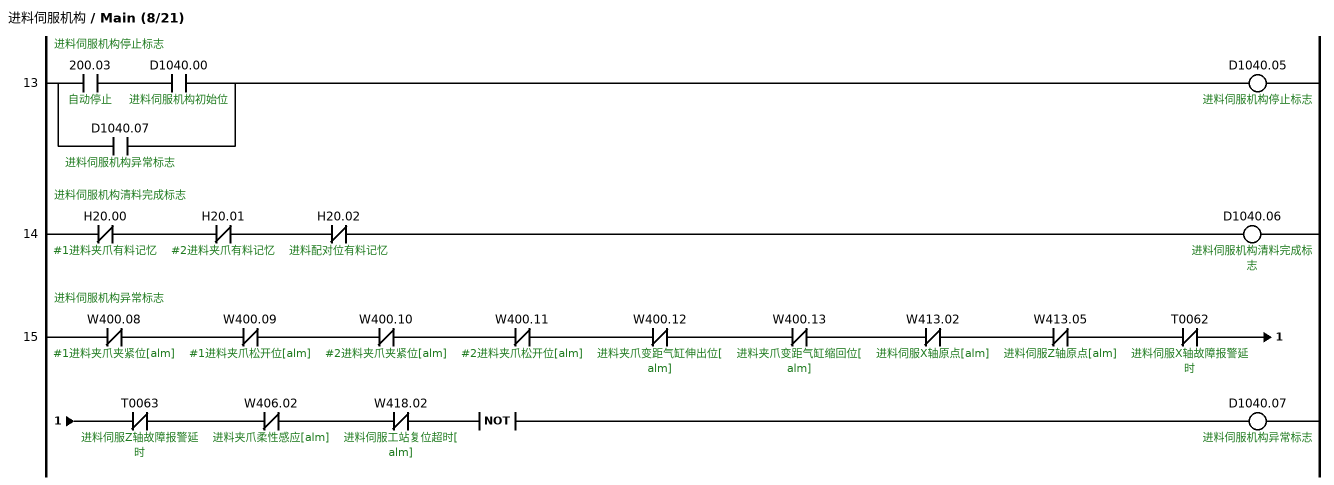
; [picture p72: 进料伺服机构 / Main, rungs 13-15]
; rung 13: 进料伺服机构停止标志
LD 200.03  ; 自动停止
AND D1040.00  ; 进料伺服机构初始位
OR D1040.07  ; 进料伺服机构异常标志
OUT D1040.05  ; 进料伺服机构停止标志
; rung 14: 进料伺服机构清料完成标志
LDNOT H20.00  ; #1进料夹爪有料记忆
ANDNOT H20.01  ; #2进料夹爪有料记忆
ANDNOT H20.02  ; 进料配对位有料记忆
OUT D1040.06  ; 进料伺服机构清料完成标志
; rung 15: 进料伺服机构异常标志
LDNOT W400.08  ; #1进料夹爪夹紧位[alm]
ANDNOT W400.09  ; #1进料夹爪松开位[alm]
ANDNOT W400.10  ; #2进料夹爪夹紧位[alm]
ANDNOT W400.11  ; #2进料夹爪松开位[alm]
ANDNOT W400.12  ; 进料夹爪变距气缸伸出位[alm]
ANDNOT W400.13  ; 进料夹爪变距气缸缩回位[alm]
ANDNOT W413.02  ; 进料伺服X轴原点[alm]
ANDNOT W413.05  ; 进料伺服Z轴原点[alm]
ANDNOT T0062  ; 进料伺服X轴故障报警延时
ANDNOT T0063  ; 进料伺服Z轴故障报警延时
ANDNOT W406.02  ; 进料夹爪柔性感应[alm]
ANDNOT W418.02  ; 进料伺服工站复位超时[alm]
NOT(520)
OUT D1040.07  ; 进料伺服机构异常标志

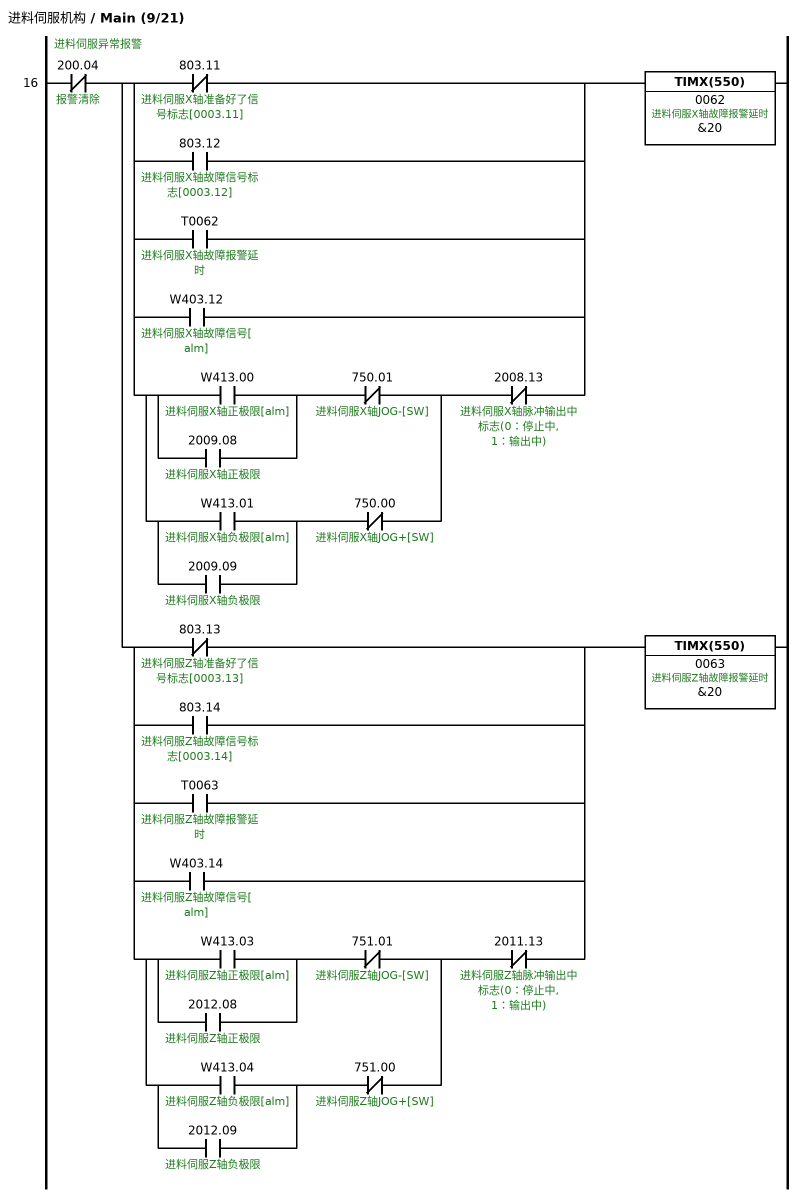
; rung 16: 进料伺服异常报警
LDNOT 200.04  ; 报警清除
OUT TR0
LDNOT 803.11  ; 进料伺服X轴准备好了信号标志[0003.11]
OR 803.12  ; 进料伺服X轴故障信号标志[0003.12]
OR T0062  ; 进料伺服X轴故障报警延时
OR W403.12  ; 进料伺服X轴故障信号[alm]
LD W413.00  ; 进料伺服X轴正极限[alm]
OR 2009.08  ; 进料伺服X轴正极限
ANDNOT 750.01  ; 进料伺服X轴JOG-[SW]
LD W413.01  ; 进料伺服X轴负极限[alm]
OR 2009.09  ; 进料伺服X轴负极限
ANDNOT 750.00  ; 进料伺服X轴JOG+[SW]
ORLD
ANDNOT 2008.13  ; 进料伺服X轴脉冲输出中标志(0：停止中,1：输出中)
ORLD
ANDLD
TIMX(550) 0062 &20  ; 进料伺服X轴故障报警延时
LD TR0
LDNOT 803.13  ; 进料伺服Z轴准备好了信号标志[0003.13]
OR 803.14  ; 进料伺服Z轴故障信号标志[0003.14]
OR T0063  ; 进料伺服Z轴故障报警延时
OR W403.14  ; 进料伺服Z轴故障信号[alm]
LD W413.03  ; 进料伺服Z轴正极限[alm]
OR 2012.08  ; 进料伺服Z轴正极限
ANDNOT 751.01  ; 进料伺服Z轴JOG-[SW]
LD W413.04  ; 进料伺服Z轴负极限[alm]
OR 2012.09  ; 进料伺服Z轴负极限
ANDNOT 751.00  ; 进料伺服Z轴JOG+[SW]
ORLD
ANDNOT 2011.13  ; 进料伺服Z轴脉冲输出中标志(0：停止中,1：输出中)
ORLD
ANDLD
TIMX(550) 0063 &20  ; 进料伺服Z轴故障报警延时

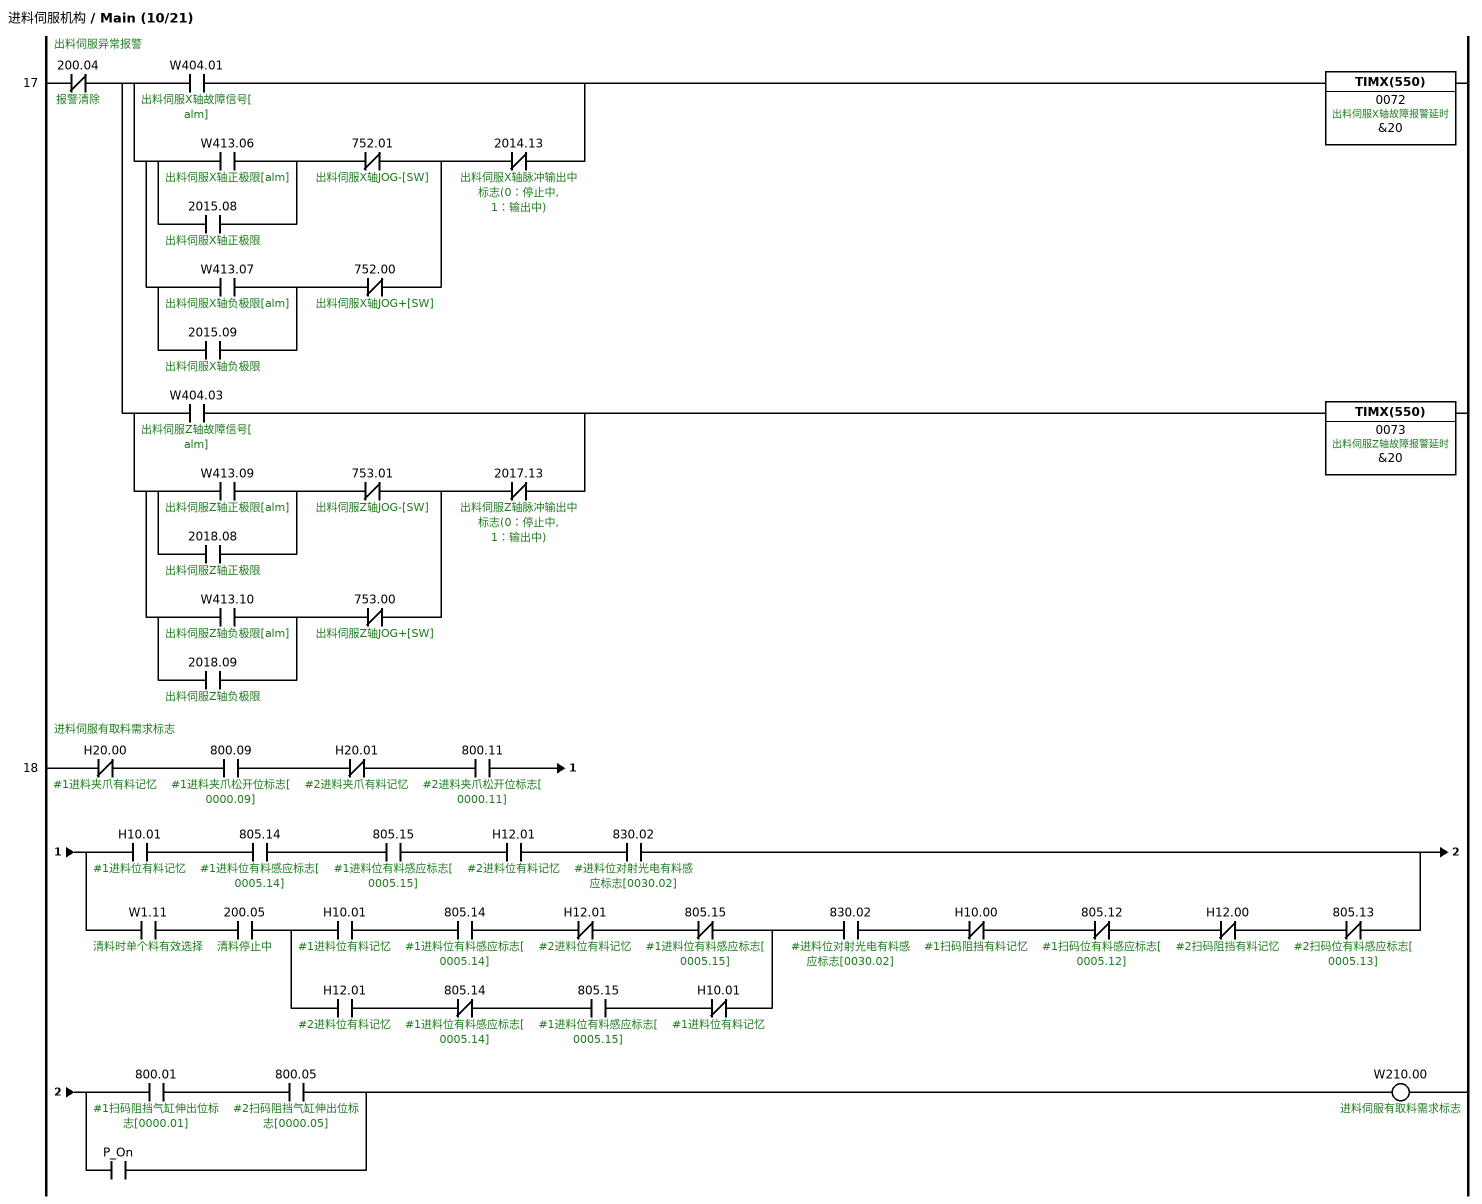
; rung 17: 出料伺服异常报警
LDNOT 200.04  ; 报警清除
OUT TR0
LD W404.01  ; 出料伺服X轴故障信号[alm]
LD W413.06  ; 出料伺服X轴正极限[alm]
OR 2015.08  ; 出料伺服X轴正极限
ANDNOT 752.01  ; 出料伺服X轴JOG-[SW]
LD W413.07  ; 出料伺服X轴负极限[alm]
OR 2015.09  ; 出料伺服X轴负极限
ANDNOT 752.00  ; 出料伺服X轴JOG+[SW]
ORLD
ANDNOT 2014.13  ; 出料伺服X轴脉冲输出中标志(0：停止中,1：输出中)
ORLD
ANDLD
TIMX(550) 0072 &20  ; 出料伺服X轴故障报警延时
LD TR0
LD W404.03  ; 出料伺服Z轴故障信号[alm]
LD W413.09  ; 出料伺服Z轴正极限[alm]
OR 2018.08  ; 出料伺服Z轴正极限
ANDNOT 753.01  ; 出料伺服Z轴JOG-[SW]
LD W413.10  ; 出料伺服Z轴负极限[alm]
OR 2018.09  ; 出料伺服Z轴负极限
ANDNOT 753.00  ; 出料伺服Z轴JOG+[SW]
ORLD
ANDNOT 2017.13  ; 出料伺服Z轴脉冲输出中标志(0：停止中,1：输出中)
ORLD
ANDLD
TIMX(550) 0073 &20  ; 出料伺服Z轴故障报警延时
; rung 18: 进料伺服有取料需求标志
LDNOT H20.00  ; #1进料夹爪有料记忆
AND 800.09  ; #1进料夹爪松开位标志[0000.09]
ANDNOT H20.01  ; #2进料夹爪有料记忆
AND 800.11  ; #2进料夹爪松开位标志[0000.11]
LD H10.01  ; #1进料位有料记忆
AND 805.14  ; #1进料位有料感应标志[0005.14]
AND 805.15  ; #1进料位有料感应标志[0005.15]
AND H12.01  ; #2进料位有料记忆
AND 830.02  ; #进料位对射光电有料感应标志[0030.02]
LD W1.11  ; 清料时单个料有效选择
AND 200.05  ; 清料停止中
LD H10.01  ; #1进料位有料记忆
AND 805.14  ; #1进料位有料感应标志[0005.14]
ANDNOT H12.01  ; #2进料位有料记忆
ANDNOT 805.15  ; #1进料位有料感应标志[0005.15]
LD H12.01  ; #2进料位有料记忆
ANDNOT 805.14  ; #1进料位有料感应标志[0005.14]
AND 805.15  ; #1进料位有料感应标志[0005.15]
ANDNOT H10.01  ; #1进料位有料记忆
ORLD
ANDLD
AND 830.02  ; #进料位对射光电有料感应标志[0030.02]
ANDNOT H10.00  ; #1扫码阻挡有料记忆
ANDNOT 805.12  ; #1扫码位有料感应标志[0005.12]
ANDNOT H12.00  ; #2扫码阻挡有料记忆
ANDNOT 805.13  ; #2扫码位有料感应标志[0005.13]
ORLD
ANDLD
LD 800.01  ; #1扫码阻挡气缸伸出位标志[0000.01]
AND 800.05  ; #2扫码阻挡气缸伸出位标志[0000.05]
OR P_On
ANDLD
OUT W210.00  ; 进料伺服有取料需求标志

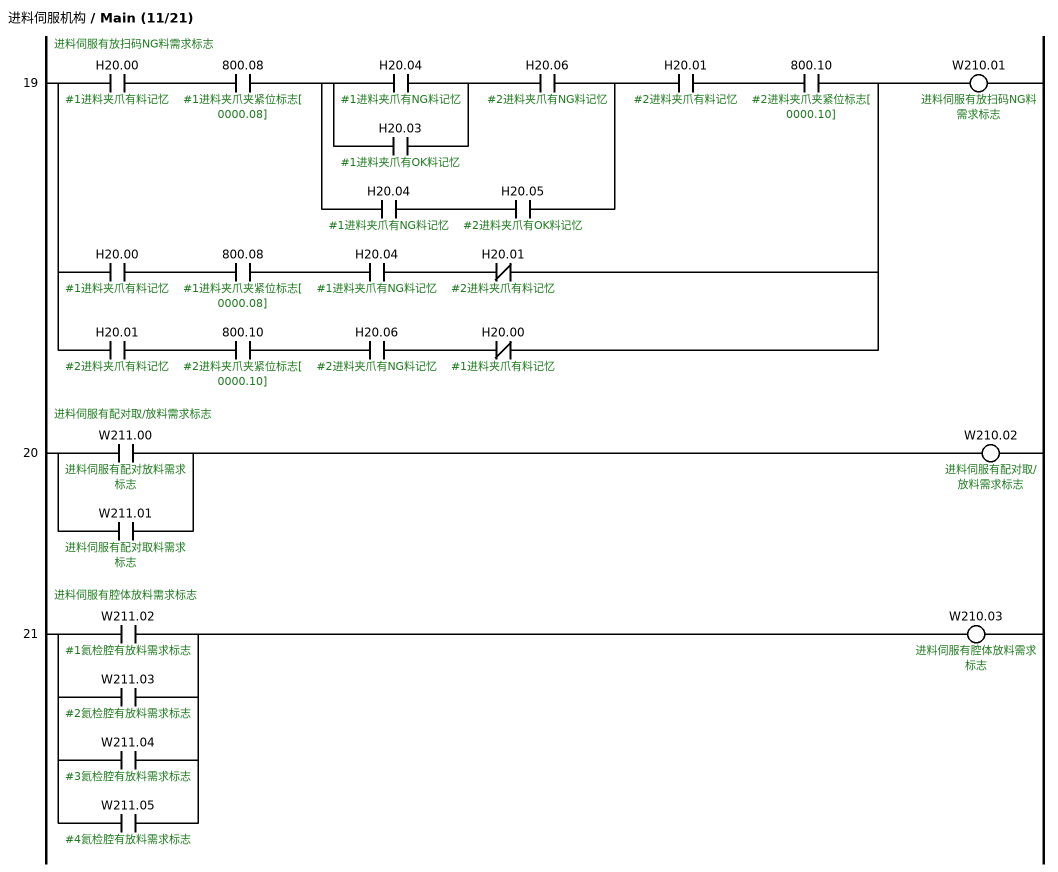
; rung 19: 进料伺服有放扫码NG料需求标志
LD H20.00  ; #1进料夹爪有料记忆
AND 800.08  ; #1进料夹爪夹紧位标志[0000.08]
LD H20.04  ; #1进料夹爪有NG料记忆
OR H20.03  ; #1进料夹爪有OK料记忆
AND H20.06  ; #2进料夹爪有NG料记忆
LD H20.04  ; #1进料夹爪有NG料记忆
AND H20.05  ; #2进料夹爪有OK料记忆
ORLD
ANDLD
AND H20.01  ; #2进料夹爪有料记忆
AND 800.10  ; #2进料夹爪夹紧位标志[0000.10]
LD H20.00  ; #1进料夹爪有料记忆
AND 800.08  ; #1进料夹爪夹紧位标志[0000.08]
AND H20.04  ; #1进料夹爪有NG料记忆
ANDNOT H20.01  ; #2进料夹爪有料记忆
ORLD
LD H20.01  ; #2进料夹爪有料记忆
AND 800.10  ; #2进料夹爪夹紧位标志[0000.10]
AND H20.06  ; #2进料夹爪有NG料记忆
ANDNOT H20.00  ; #1进料夹爪有料记忆
ORLD
OUT W210.01  ; 进料伺服有放扫码NG料需求标志
; rung 20: 进料伺服有配对取/放料需求标志
LD W211.00  ; 进料伺服有配对放料需求标志
OR W211.01  ; 进料伺服有配对取料需求标志
OUT W210.02  ; 进料伺服有配对取/放料需求标志
; rung 21: 进料伺服有腔体放料需求标志
LD W211.02  ; #1氦检腔有放料需求标志
OR W211.03  ; #2氦检腔有放料需求标志
OR W211.04  ; #3氦检腔有放料需求标志
OR W211.05  ; #4氦检腔有放料需求标志
OUT W210.03  ; 进料伺服有腔体放料需求标志

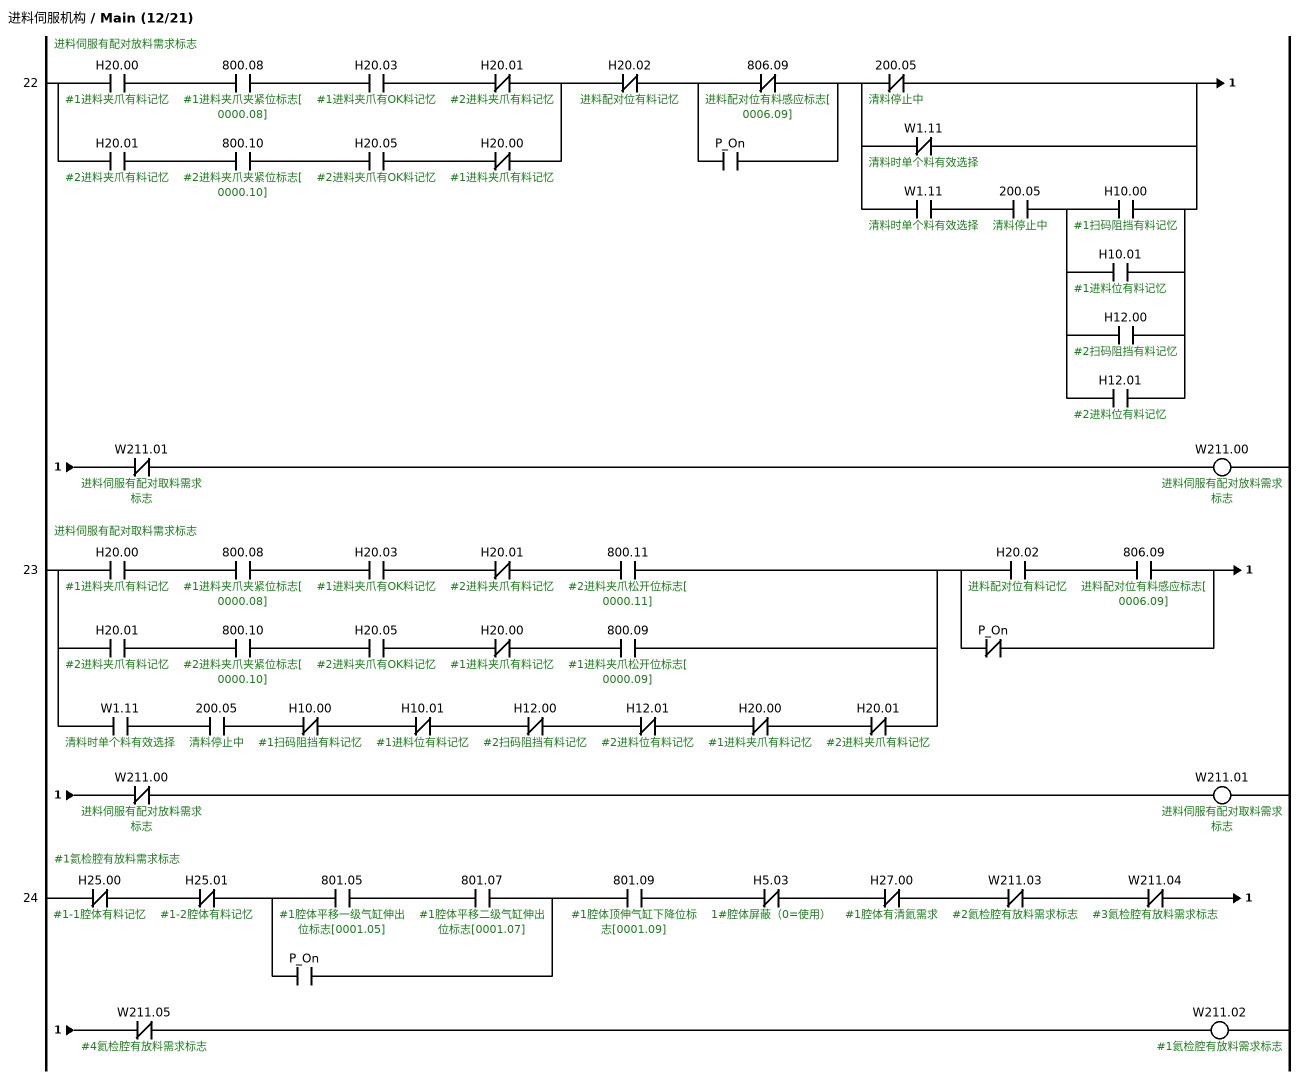
; rung 22: 进料伺服有配对放料需求标志
LD H20.00  ; #1进料夹爪有料记忆
AND 800.08  ; #1进料夹爪夹紧位标志[0000.08]
AND H20.03  ; #1进料夹爪有OK料记忆
ANDNOT H20.01  ; #2进料夹爪有料记忆
LD H20.01  ; #2进料夹爪有料记忆
AND 800.10  ; #2进料夹爪夹紧位标志[0000.10]
AND H20.05  ; #2进料夹爪有OK料记忆
ANDNOT H20.00  ; #1进料夹爪有料记忆
ORLD
ANDNOT H20.02  ; 进料配对位有料记忆
LDNOT 806.09  ; 进料配对位有料感应标志[0006.09]
OR P_On
ANDLD
LDNOT 200.05  ; 清料停止中
ORNOT W1.11  ; 清料时单个料有效选择
LD W1.11  ; 清料时单个料有效选择
AND 200.05  ; 清料停止中
LD H10.00  ; #1扫码阻挡有料记忆
OR H10.01  ; #1进料位有料记忆
OR H12.00  ; #2扫码阻挡有料记忆
OR H12.01  ; #2进料位有料记忆
ANDLD
ORLD
ANDLD
ANDNOT W211.01  ; 进料伺服有配对取料需求标志
OUT W211.00  ; 进料伺服有配对放料需求标志
; rung 23: 进料伺服有配对取料需求标志
LD H20.00  ; #1进料夹爪有料记忆
AND 800.08  ; #1进料夹爪夹紧位标志[0000.08]
AND H20.03  ; #1进料夹爪有OK料记忆
ANDNOT H20.01  ; #2进料夹爪有料记忆
AND 800.11  ; #2进料夹爪松开位标志[0000.11]
LD H20.01  ; #2进料夹爪有料记忆
AND 800.10  ; #2进料夹爪夹紧位标志[0000.10]
AND H20.05  ; #2进料夹爪有OK料记忆
ANDNOT H20.00  ; #1进料夹爪有料记忆
AND 800.09  ; #1进料夹爪松开位标志[0000.09]
ORLD
LD W1.11  ; 清料时单个料有效选择
AND 200.05  ; 清料停止中
ANDNOT H10.00  ; #1扫码阻挡有料记忆
ANDNOT H10.01  ; #1进料位有料记忆
ANDNOT H12.00  ; #2扫码阻挡有料记忆
ANDNOT H12.01  ; #2进料位有料记忆
ANDNOT H20.00  ; #1进料夹爪有料记忆
ANDNOT H20.01  ; #2进料夹爪有料记忆
ORLD
LD H20.02  ; 进料配对位有料记忆
AND 806.09  ; 进料配对位有料感应标志[0006.09]
ORNOT P_On
ANDLD
ANDNOT W211.00  ; 进料伺服有配对放料需求标志
OUT W211.01  ; 进料伺服有配对取料需求标志
; rung 24: #1氦检腔有放料需求标志
LDNOT H25.00  ; #1-1腔体有料记忆
ANDNOT H25.01  ; #1-2腔体有料记忆
LD 801.05  ; #1腔体平移一级气缸伸出位标志[0001.05]
AND 801.07  ; #1腔体平移二级气缸伸出位标志[0001.07]
OR P_On
ANDLD
AND 801.09  ; #1腔体顶伸气缸下降位标志[0001.09]
ANDNOT H5.03  ; 1#腔体屏蔽（0=使用）
ANDNOT H27.00  ; #1腔体有清氦需求
ANDNOT W211.03  ; #2氦检腔有放料需求标志
ANDNOT W211.04  ; #3氦检腔有放料需求标志
ANDNOT W211.05  ; #4氦检腔有放料需求标志
OUT W211.02  ; #1氦检腔有放料需求标志

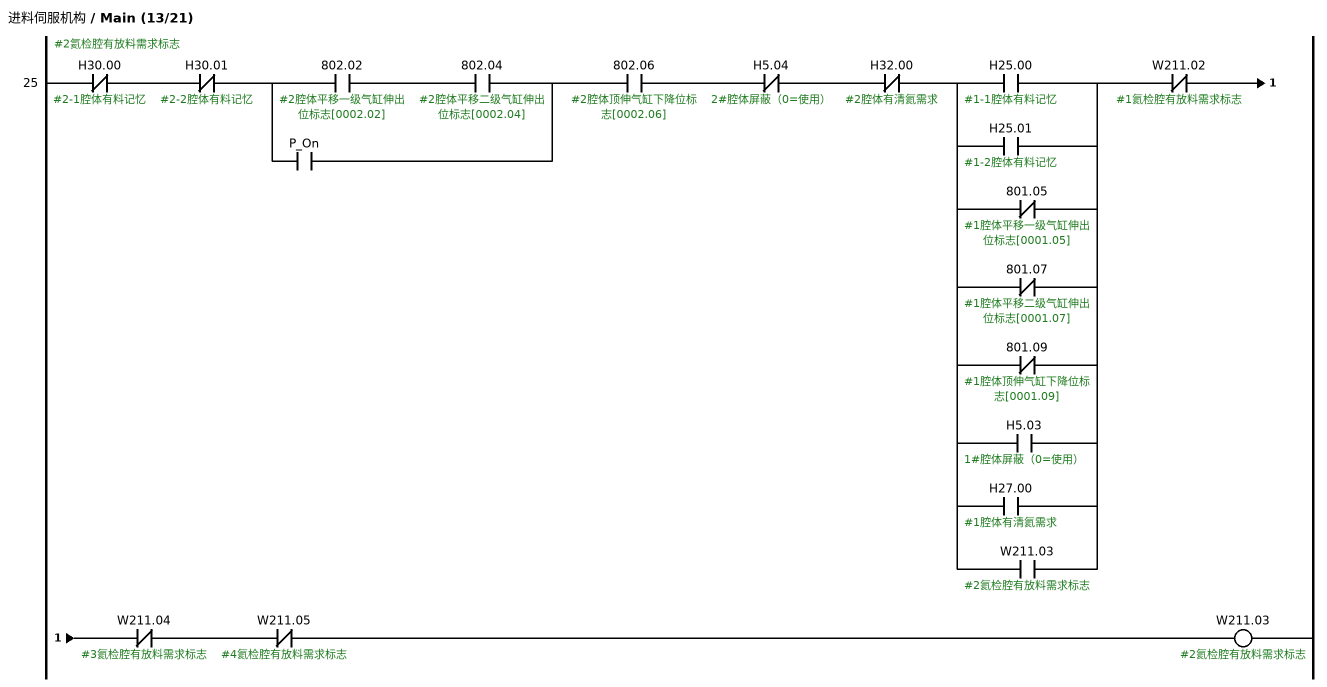
; rung 25: #2氦检腔有放料需求标志
LDNOT H30.00  ; #2-1腔体有料记忆
ANDNOT H30.01  ; #2-2腔体有料记忆
LD 802.02  ; #2腔体平移一级气缸伸出位标志[0002.02]
AND 802.04  ; #2腔体平移二级气缸伸出位标志[0002.04]
OR P_On
ANDLD
AND 802.06  ; #2腔体顶伸气缸下降位标志[0002.06]
ANDNOT H5.04  ; 2#腔体屏蔽（0=使用）
ANDNOT H32.00  ; #2腔体有清氦需求
LD H25.00  ; #1-1腔体有料记忆
OR H25.01  ; #1-2腔体有料记忆
ORNOT 801.05  ; #1腔体平移一级气缸伸出位标志[0001.05]
ORNOT 801.07  ; #1腔体平移二级气缸伸出位标志[0001.07]
ORNOT 801.09  ; #1腔体顶伸气缸下降位标志[0001.09]
OR H5.03  ; 1#腔体屏蔽（0=使用）
OR H27.00  ; #1腔体有清氦需求
OR W211.03  ; #2氦检腔有放料需求标志
ANDLD
ANDNOT W211.02  ; #1氦检腔有放料需求标志
ANDNOT W211.04  ; #3氦检腔有放料需求标志
ANDNOT W211.05  ; #4氦检腔有放料需求标志
OUT W211.03  ; #2氦检腔有放料需求标志

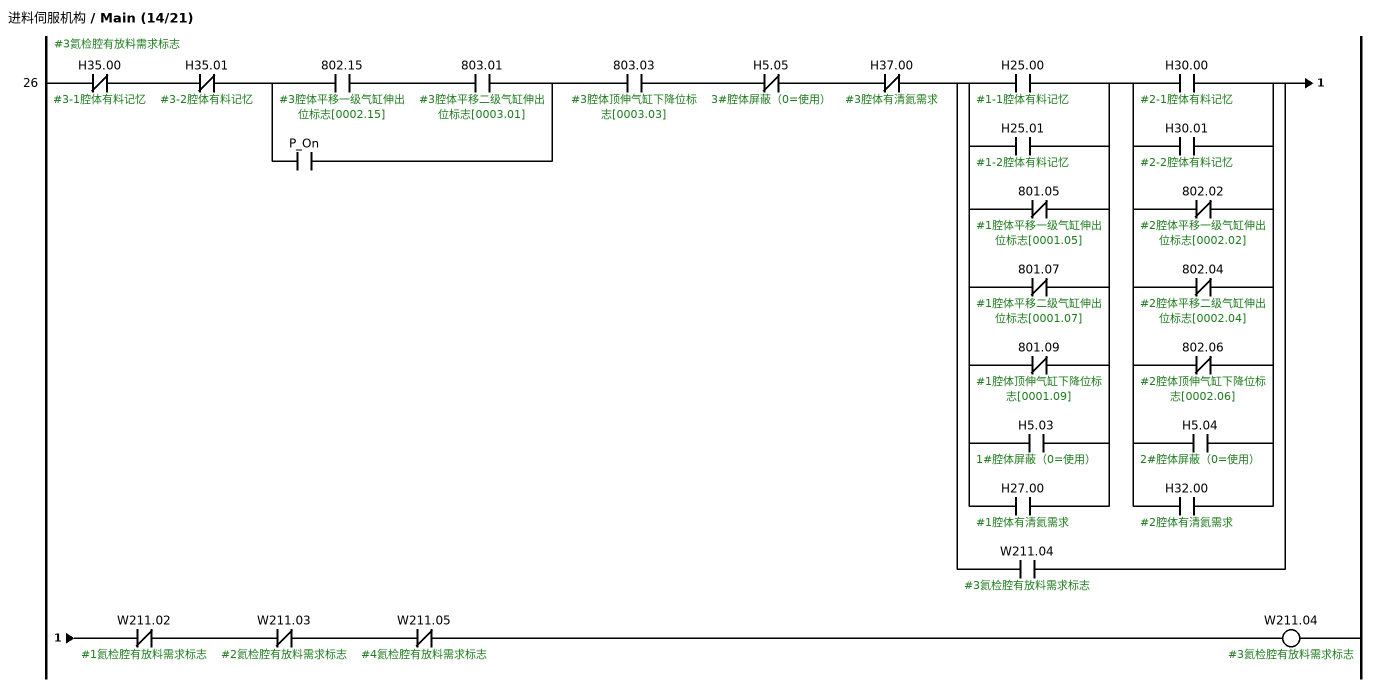
; rung 26: #3氦检腔有放料需求标志
LDNOT H35.00  ; #3-1腔体有料记忆
ANDNOT H35.01  ; #3-2腔体有料记忆
LD 802.15  ; #3腔体平移一级气缸伸出位标志[0002.15]
AND 803.01  ; #3腔体平移二级气缸伸出位标志[0003.01]
OR P_On
ANDLD
AND 803.03  ; #3腔体顶伸气缸下降位标志[0003.03]
ANDNOT H5.05  ; 3#腔体屏蔽（0=使用）
ANDNOT H37.00  ; #3腔体有清氦需求
LD H25.00  ; #1-1腔体有料记忆
OR H25.01  ; #1-2腔体有料记忆
ORNOT 801.05  ; #1腔体平移一级气缸伸出位标志[0001.05]
ORNOT 801.07  ; #1腔体平移二级气缸伸出位标志[0001.07]
ORNOT 801.09  ; #1腔体顶伸气缸下降位标志[0001.09]
OR H5.03  ; 1#腔体屏蔽（0=使用）
OR H27.00  ; #1腔体有清氦需求
LD H30.00  ; #2-1腔体有料记忆
OR H30.01  ; #2-2腔体有料记忆
ORNOT 802.02  ; #2腔体平移一级气缸伸出位标志[0002.02]
ORNOT 802.04  ; #2腔体平移二级气缸伸出位标志[0002.04]
ORNOT 802.06  ; #2腔体顶伸气缸下降位标志[0002.06]
OR H5.04  ; 2#腔体屏蔽（0=使用）
OR H32.00  ; #2腔体有清氦需求
ANDLD
OR W211.04  ; #3氦检腔有放料需求标志
ANDLD
ANDNOT W211.02  ; #1氦检腔有放料需求标志
ANDNOT W211.03  ; #2氦检腔有放料需求标志
ANDNOT W211.05  ; #4氦检腔有放料需求标志
OUT W211.04  ; #3氦检腔有放料需求标志

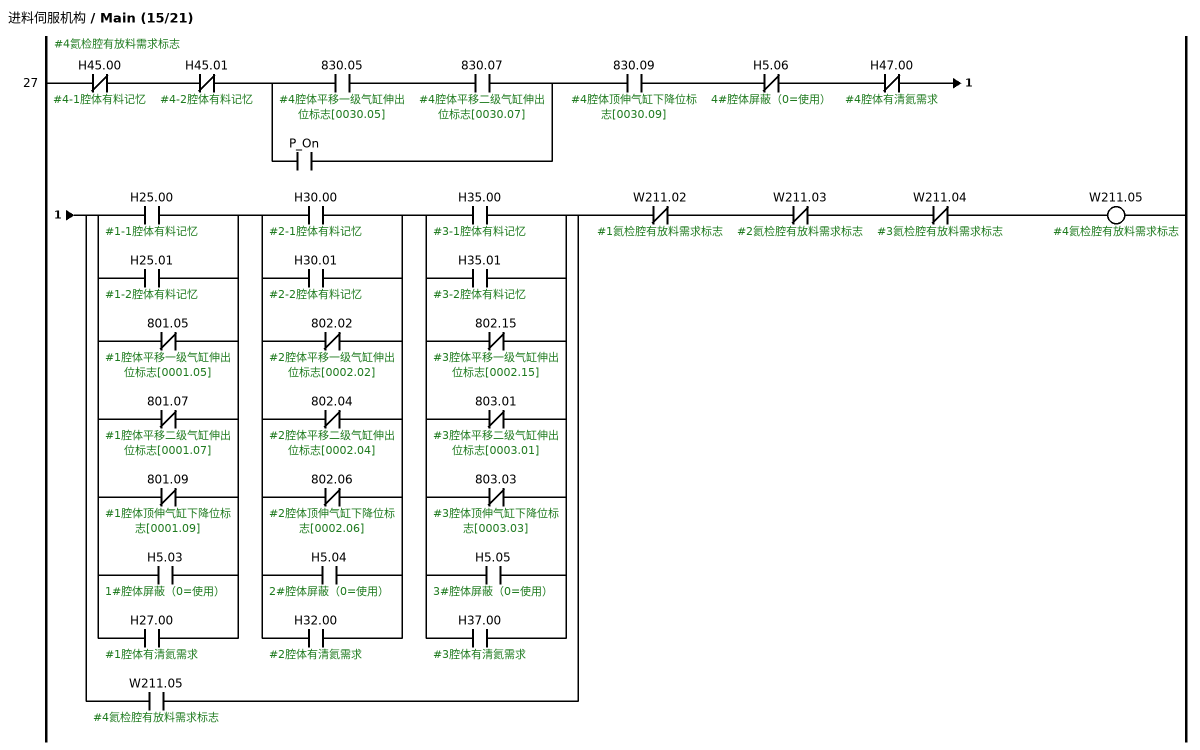
; rung 27: #4氦检腔有放料需求标志
LDNOT H45.00  ; #4-1腔体有料记忆
ANDNOT H45.01  ; #4-2腔体有料记忆
LD 830.05  ; #4腔体平移一级气缸伸出位标志[0030.05]
AND 830.07  ; #4腔体平移二级气缸伸出位标志[0030.07]
OR P_On
ANDLD
AND 830.09  ; #4腔体顶伸气缸下降位标志[0030.09]
ANDNOT H5.06  ; 4#腔体屏蔽（0=使用）
ANDNOT H47.00  ; #4腔体有清氦需求
LD H25.00  ; #1-1腔体有料记忆
OR H25.01  ; #1-2腔体有料记忆
ORNOT 801.05  ; #1腔体平移一级气缸伸出位标志[0001.05]
ORNOT 801.07  ; #1腔体平移二级气缸伸出位标志[0001.07]
ORNOT 801.09  ; #1腔体顶伸气缸下降位标志[0001.09]
OR H5.03  ; 1#腔体屏蔽（0=使用）
OR H27.00  ; #1腔体有清氦需求
LD H30.00  ; #2-1腔体有料记忆
OR H30.01  ; #2-2腔体有料记忆
ORNOT 802.02  ; #2腔体平移一级气缸伸出位标志[0002.02]
ORNOT 802.04  ; #2腔体平移二级气缸伸出位标志[0002.04]
ORNOT 802.06  ; #2腔体顶伸气缸下降位标志[0002.06]
OR H5.04  ; 2#腔体屏蔽（0=使用）
OR H32.00  ; #2腔体有清氦需求
ANDLD
LD H35.00  ; #3-1腔体有料记忆
OR H35.01  ; #3-2腔体有料记忆
ORNOT 802.15  ; #3腔体平移一级气缸伸出位标志[0002.15]
ORNOT 803.01  ; #3腔体平移二级气缸伸出位标志[0003.01]
ORNOT 803.03  ; #3腔体顶伸气缸下降位标志[0003.03]
OR H5.05  ; 3#腔体屏蔽（0=使用）
OR H37.00  ; #3腔体有清氦需求
ANDLD
OR W211.05  ; #4氦检腔有放料需求标志
ANDLD
ANDNOT W211.02  ; #1氦检腔有放料需求标志
ANDNOT W211.03  ; #2氦检腔有放料需求标志
ANDNOT W211.04  ; #3氦检腔有放料需求标志
OUT W211.05  ; #4氦检腔有放料需求标志

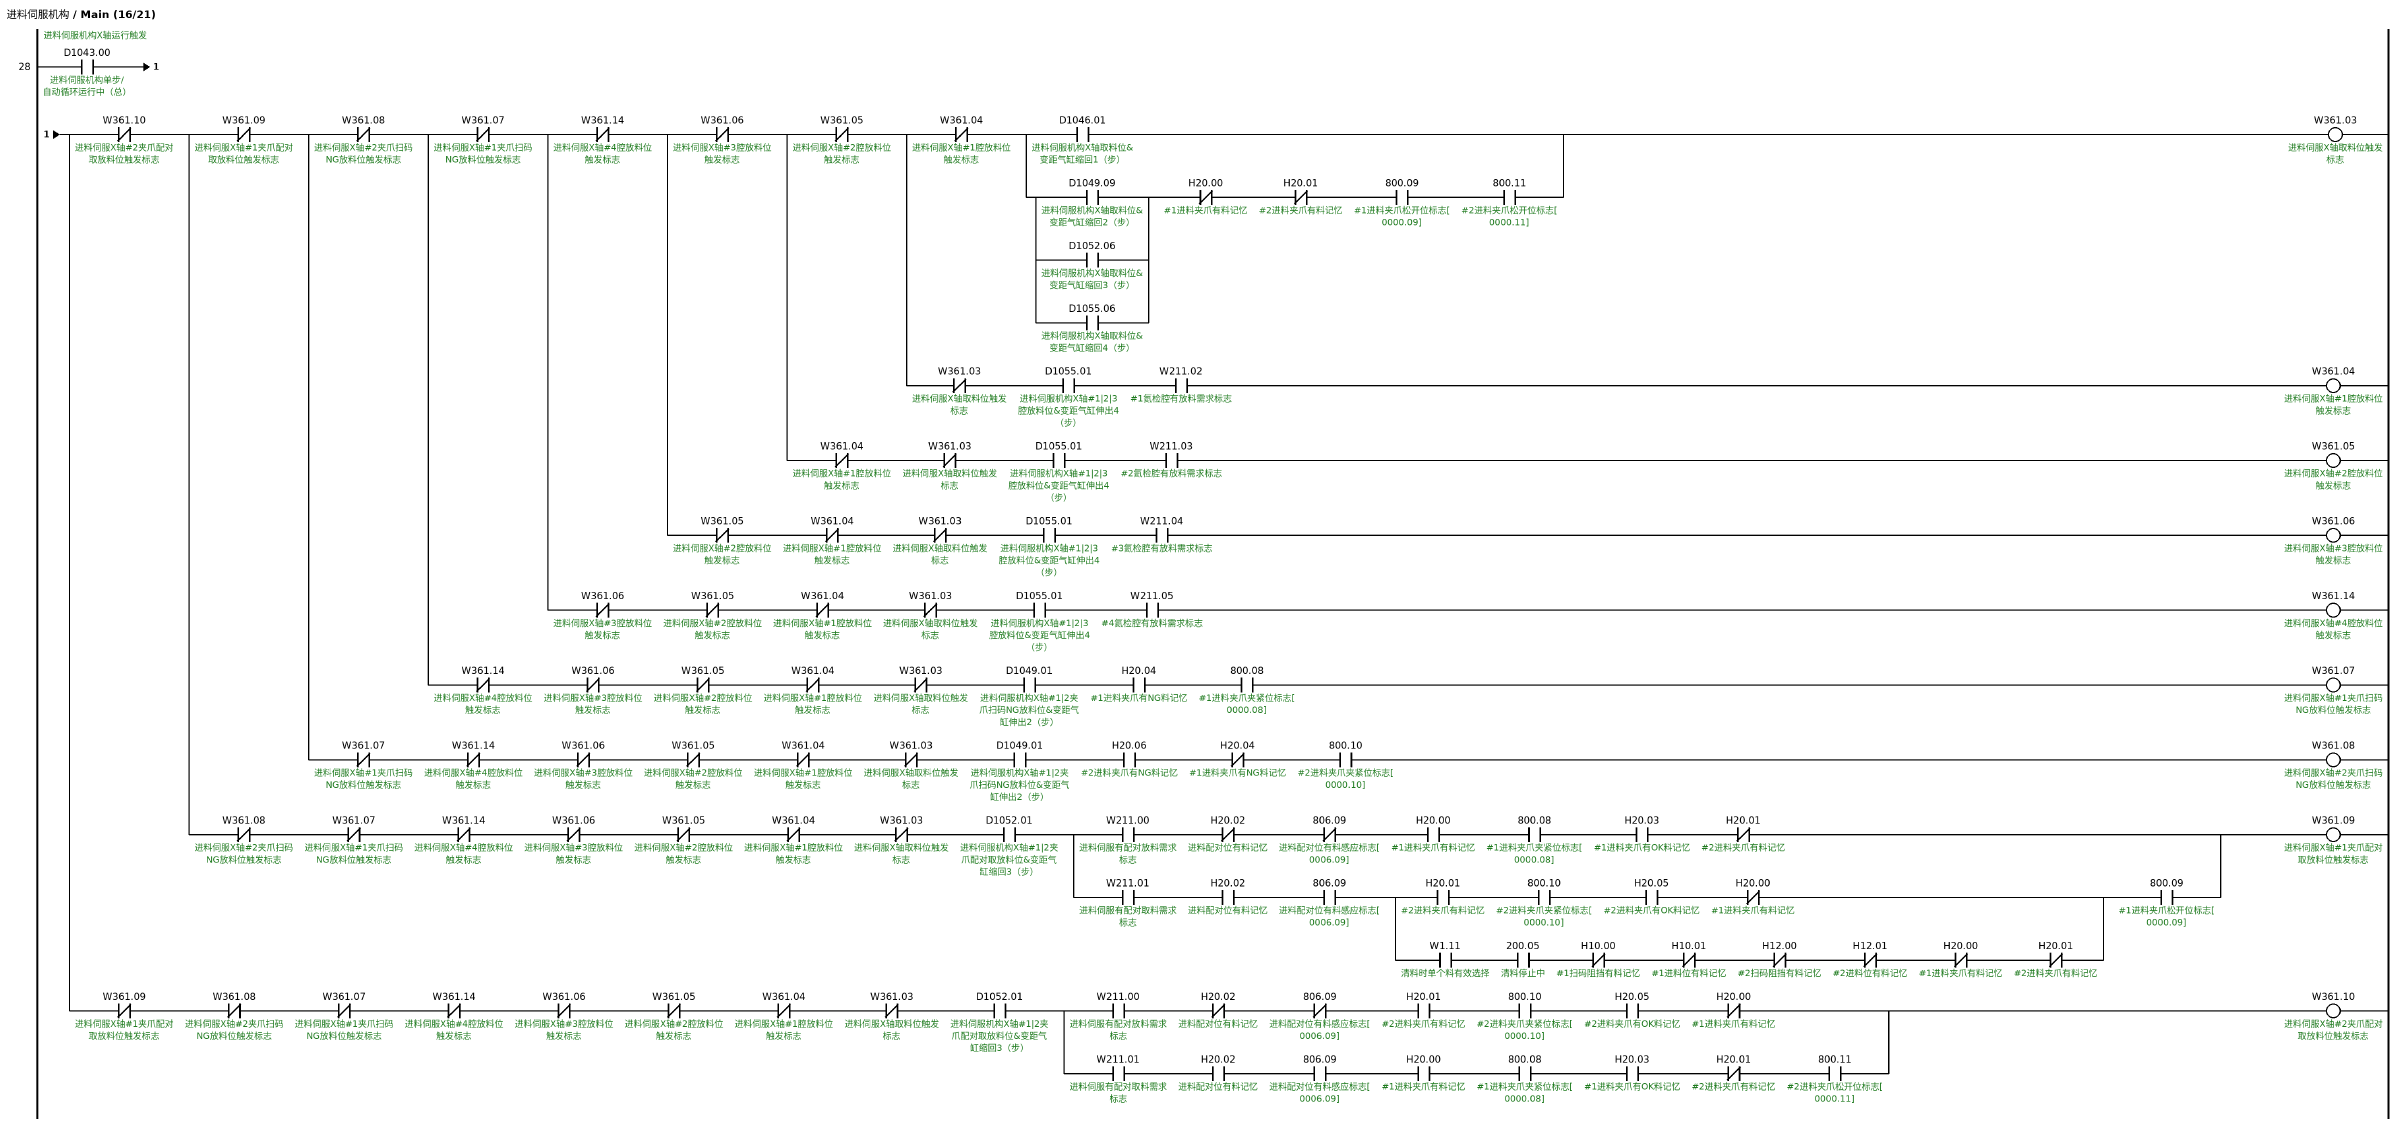
; rung 28: 进料伺服机构X轴运行触发
LD D1043.00  ; 进料伺服机构单步/自动循环运行中（总）
OUT TR0
ANDNOT W361.10  ; 进料伺服X轴#2夹爪配对取放料位触发标志
OUT TR1
ANDNOT W361.09  ; 进料伺服X轴#1夹爪配对取放料位触发标志
OUT TR2
ANDNOT W361.08  ; 进料伺服X轴#2夹爪扫码NG放料位触发标志
OUT TR3
ANDNOT W361.07  ; 进料伺服X轴#1夹爪扫码NG放料位触发标志
OUT TR4
ANDNOT W361.14  ; 进料伺服X轴#4腔放料位触发标志
OUT TR5
ANDNOT W361.06  ; 进料伺服X轴#3腔放料位触发标志
OUT TR6
ANDNOT W361.05  ; 进料伺服X轴#2腔放料位触发标志
OUT TR7
ANDNOT W361.04  ; 进料伺服X轴#1腔放料位触发标志
LD D1046.01  ; 进料伺服机构X轴取料位&变距气缸缩回1（步）
LD D1049.09  ; 进料伺服机构X轴取料位&变距气缸缩回2（步）
OR D1052.06  ; 进料伺服机构X轴取料位&变距气缸缩回3（步）
OR D1055.06  ; 进料伺服机构X轴取料位&变距气缸缩回4（步）
ANDNOT H20.00  ; #1进料夹爪有料记忆
ANDNOT H20.01  ; #2进料夹爪有料记忆
AND 800.09  ; #1进料夹爪松开位标志[0000.09]
AND 800.11  ; #2进料夹爪松开位标志[0000.11]
ORLD
ANDLD
OUT W361.03  ; 进料伺服X轴取料位触发标志
LD TR7
ANDNOT W361.03  ; 进料伺服X轴取料位触发标志
AND D1055.01  ; 进料伺服机构X轴#1|2|3腔放料位&变距气缸伸出4（步）
AND W211.02  ; #1氦检腔有放料需求标志
OUT W361.04  ; 进料伺服X轴#1腔放料位触发标志
LD TR6
ANDNOT W361.04  ; 进料伺服X轴#1腔放料位触发标志
ANDNOT W361.03  ; 进料伺服X轴取料位触发标志
AND D1055.01  ; 进料伺服机构X轴#1|2|3腔放料位&变距气缸伸出4（步）
AND W211.03  ; #2氦检腔有放料需求标志
OUT W361.05  ; 进料伺服X轴#2腔放料位触发标志
LD TR5
ANDNOT W361.05  ; 进料伺服X轴#2腔放料位触发标志
ANDNOT W361.04  ; 进料伺服X轴#1腔放料位触发标志
ANDNOT W361.03  ; 进料伺服X轴取料位触发标志
AND D1055.01  ; 进料伺服机构X轴#1|2|3腔放料位&变距气缸伸出4（步）
AND W211.04  ; #3氦检腔有放料需求标志
OUT W361.06  ; 进料伺服X轴#3腔放料位触发标志
LD TR4
ANDNOT W361.06  ; 进料伺服X轴#3腔放料位触发标志
ANDNOT W361.05  ; 进料伺服X轴#2腔放料位触发标志
ANDNOT W361.04  ; 进料伺服X轴#1腔放料位触发标志
ANDNOT W361.03  ; 进料伺服X轴取料位触发标志
AND D1055.01  ; 进料伺服机构X轴#1|2|3腔放料位&变距气缸伸出4（步）
AND W211.05  ; #4氦检腔有放料需求标志
OUT W361.14  ; 进料伺服X轴#4腔放料位触发标志
LD TR3
ANDNOT W361.14  ; 进料伺服X轴#4腔放料位触发标志
ANDNOT W361.06  ; 进料伺服X轴#3腔放料位触发标志
ANDNOT W361.05  ; 进料伺服X轴#2腔放料位触发标志
ANDNOT W361.04  ; 进料伺服X轴#1腔放料位触发标志
ANDNOT W361.03  ; 进料伺服X轴取料位触发标志
AND D1049.01  ; 进料伺服机构X轴#1|2夹爪扫码NG放料位&变距气缸伸出2（步）
AND H20.04  ; #1进料夹爪有NG料记忆
AND 800.08  ; #1进料夹爪夹紧位标志[0000.08]
OUT W361.07  ; 进料伺服X轴#1夹爪扫码NG放料位触发标志
LD TR2
ANDNOT W361.07  ; 进料伺服X轴#1夹爪扫码NG放料位触发标志
ANDNOT W361.14  ; 进料伺服X轴#4腔放料位触发标志
ANDNOT W361.06  ; 进料伺服X轴#3腔放料位触发标志
ANDNOT W361.05  ; 进料伺服X轴#2腔放料位触发标志
ANDNOT W361.04  ; 进料伺服X轴#1腔放料位触发标志
ANDNOT W361.03  ; 进料伺服X轴取料位触发标志
AND D1049.01  ; 进料伺服机构X轴#1|2夹爪扫码NG放料位&变距气缸伸出2（步）
AND H20.06  ; #2进料夹爪有NG料记忆
ANDNOT H20.04  ; #1进料夹爪有NG料记忆
AND 800.10  ; #2进料夹爪夹紧位标志[0000.10]
OUT W361.08  ; 进料伺服X轴#2夹爪扫码NG放料位触发标志
LD TR1
ANDNOT W361.08  ; 进料伺服X轴#2夹爪扫码NG放料位触发标志
ANDNOT W361.07  ; 进料伺服X轴#1夹爪扫码NG放料位触发标志
ANDNOT W361.14  ; 进料伺服X轴#4腔放料位触发标志
ANDNOT W361.06  ; 进料伺服X轴#3腔放料位触发标志
ANDNOT W361.05  ; 进料伺服X轴#2腔放料位触发标志
ANDNOT W361.04  ; 进料伺服X轴#1腔放料位触发标志
ANDNOT W361.03  ; 进料伺服X轴取料位触发标志
AND D1052.01  ; 进料伺服机构X轴#1|2夹爪配对取放料位&变距气缸缩回3（步）
LD W211.00  ; 进料伺服有配对放料需求标志
ANDNOT H20.02  ; 进料配对位有料记忆
ANDNOT 806.09  ; 进料配对位有料感应标志[0006.09]
AND H20.00  ; #1进料夹爪有料记忆
AND 800.08  ; #1进料夹爪夹紧位标志[0000.08]
AND H20.03  ; #1进料夹爪有OK料记忆
ANDNOT H20.01  ; #2进料夹爪有料记忆
LD W211.01  ; 进料伺服有配对取料需求标志
AND H20.02  ; 进料配对位有料记忆
AND 806.09  ; 进料配对位有料感应标志[0006.09]
LD H20.01  ; #2进料夹爪有料记忆
AND 800.10  ; #2进料夹爪夹紧位标志[0000.10]
AND H20.05  ; #2进料夹爪有OK料记忆
ANDNOT H20.00  ; #1进料夹爪有料记忆
LD W1.11  ; 清料时单个料有效选择
AND 200.05  ; 清料停止中
ANDNOT H10.00  ; #1扫码阻挡有料记忆
ANDNOT H10.01  ; #1进料位有料记忆
ANDNOT H12.00  ; #2扫码阻挡有料记忆
ANDNOT H12.01  ; #2进料位有料记忆
ANDNOT H20.00  ; #1进料夹爪有料记忆
ANDNOT H20.01  ; #2进料夹爪有料记忆
ORLD
ANDLD
AND 800.09  ; #1进料夹爪松开位标志[0000.09]
ORLD
ANDLD
OUT W361.09  ; 进料伺服X轴#1夹爪配对取放料位触发标志
LD TR0
ANDNOT W361.09  ; 进料伺服X轴#1夹爪配对取放料位触发标志
ANDNOT W361.08  ; 进料伺服X轴#2夹爪扫码NG放料位触发标志
ANDNOT W361.07  ; 进料伺服X轴#1夹爪扫码NG放料位触发标志
ANDNOT W361.14  ; 进料伺服X轴#4腔放料位触发标志
ANDNOT W361.06  ; 进料伺服X轴#3腔放料位触发标志
ANDNOT W361.05  ; 进料伺服X轴#2腔放料位触发标志
ANDNOT W361.04  ; 进料伺服X轴#1腔放料位触发标志
ANDNOT W361.03  ; 进料伺服X轴取料位触发标志
AND D1052.01  ; 进料伺服机构X轴#1|2夹爪配对取放料位&变距气缸缩回3（步）
LD W211.00  ; 进料伺服有配对放料需求标志
ANDNOT H20.02  ; 进料配对位有料记忆
ANDNOT 806.09  ; 进料配对位有料感应标志[0006.09]
AND H20.01  ; #2进料夹爪有料记忆
AND 800.10  ; #2进料夹爪夹紧位标志[0000.10]
AND H20.05  ; #2进料夹爪有OK料记忆
ANDNOT H20.00  ; #1进料夹爪有料记忆
LD W211.01  ; 进料伺服有配对取料需求标志
AND H20.02  ; 进料配对位有料记忆
AND 806.09  ; 进料配对位有料感应标志[0006.09]
AND H20.00  ; #1进料夹爪有料记忆
AND 800.08  ; #1进料夹爪夹紧位标志[0000.08]
AND H20.03  ; #1进料夹爪有OK料记忆
ANDNOT H20.01  ; #2进料夹爪有料记忆
AND 800.11  ; #2进料夹爪松开位标志[0000.11]
ORLD
ANDLD
OUT W361.10  ; 进料伺服X轴#2夹爪配对取放料位触发标志

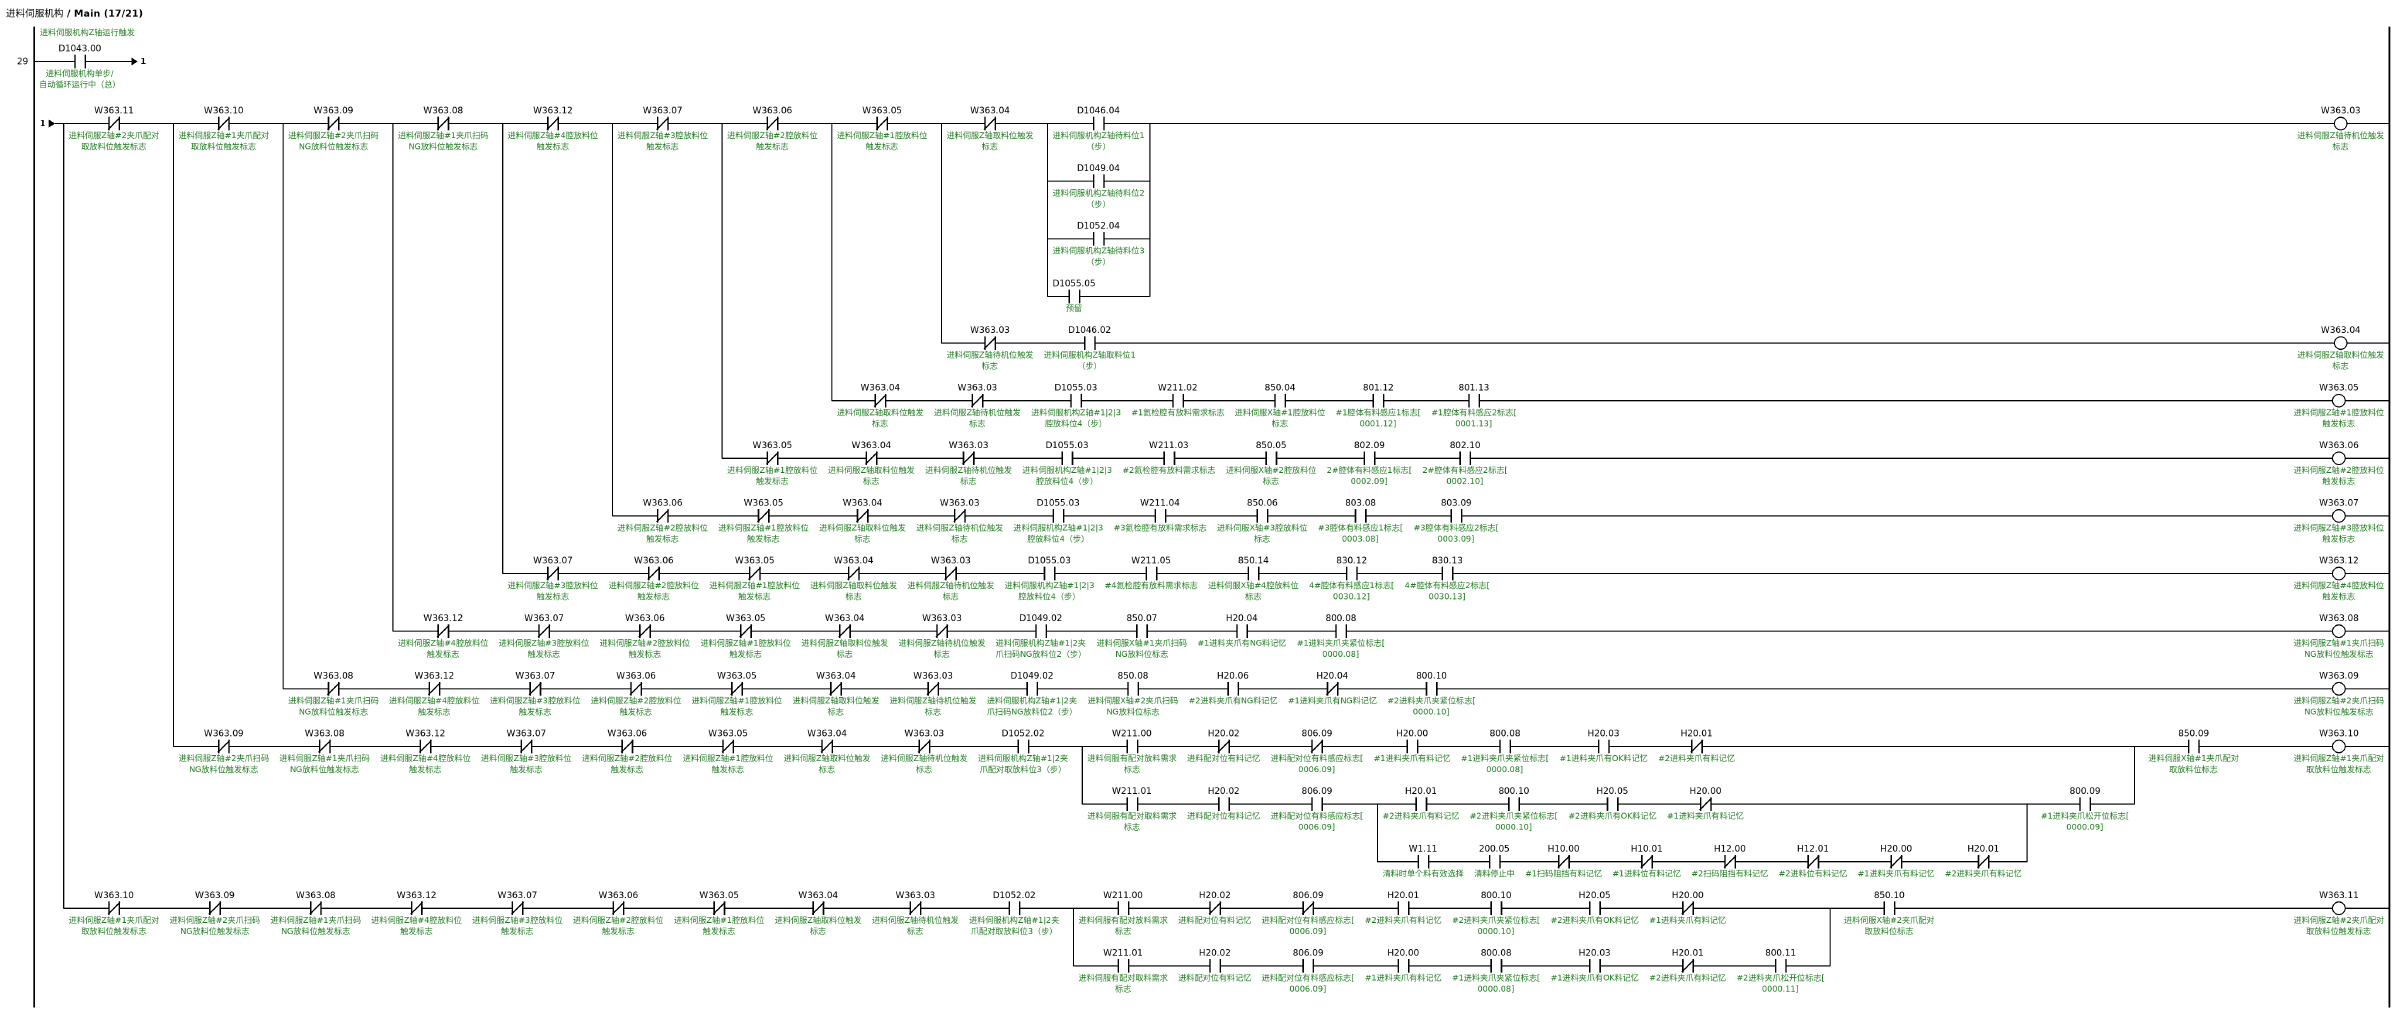
; rung 29: 进料伺服机构Z轴运行触发
LD D1043.00  ; 进料伺服机构单步/自动循环运行中（总）
OUT TR0
ANDNOT W363.11  ; 进料伺服Z轴#2夹爪配对取放料位触发标志
OUT TR1
ANDNOT W363.10  ; 进料伺服Z轴#1夹爪配对取放料位触发标志
OUT TR2
ANDNOT W363.09  ; 进料伺服Z轴#2夹爪扫码NG放料位触发标志
OUT TR3
ANDNOT W363.08  ; 进料伺服Z轴#1夹爪扫码NG放料位触发标志
OUT TR4
ANDNOT W363.12  ; 进料伺服Z轴#4腔放料位触发标志
OUT TR5
ANDNOT W363.07  ; 进料伺服Z轴#3腔放料位触发标志
OUT TR6
ANDNOT W363.06  ; 进料伺服Z轴#2腔放料位触发标志
OUT TR7
ANDNOT W363.05  ; 进料伺服Z轴#1腔放料位触发标志
OUT TR8
ANDNOT W363.04  ; 进料伺服Z轴取料位触发标志
LD D1046.04  ; 进料伺服机构Z轴待料位1（步）
OR D1049.04  ; 进料伺服机构Z轴待料位2（步）
OR D1052.04  ; 进料伺服机构Z轴待料位3（步）
OR D1055.05  ; 预留
ANDLD
OUT W363.03  ; 进料伺服Z轴待机位触发标志
LD TR8
ANDNOT W363.03  ; 进料伺服Z轴待机位触发标志
AND D1046.02  ; 进料伺服机构Z轴取料位1（步）
OUT W363.04  ; 进料伺服Z轴取料位触发标志
LD TR7
ANDNOT W363.04  ; 进料伺服Z轴取料位触发标志
ANDNOT W363.03  ; 进料伺服Z轴待机位触发标志
AND D1055.03  ; 进料伺服机构Z轴#1|2|3腔放料位4（步）
AND W211.02  ; #1氦检腔有放料需求标志
AND 850.04  ; 进料伺服X轴#1腔放料位标志
AND 801.12  ; #1腔体有料感应1标志[0001.12]
AND 801.13  ; #1腔体有料感应2标志[0001.13]
OUT W363.05  ; 进料伺服Z轴#1腔放料位触发标志
LD TR6
ANDNOT W363.05  ; 进料伺服Z轴#1腔放料位触发标志
ANDNOT W363.04  ; 进料伺服Z轴取料位触发标志
ANDNOT W363.03  ; 进料伺服Z轴待机位触发标志
AND D1055.03  ; 进料伺服机构Z轴#1|2|3腔放料位4（步）
AND W211.03  ; #2氦检腔有放料需求标志
AND 850.05  ; 进料伺服X轴#2腔放料位标志
AND 802.09  ; 2#腔体有料感应1标志[0002.09]
AND 802.10  ; 2#腔体有料感应2标志[0002.10]
OUT W363.06  ; 进料伺服Z轴#2腔放料位触发标志
LD TR5
ANDNOT W363.06  ; 进料伺服Z轴#2腔放料位触发标志
ANDNOT W363.05  ; 进料伺服Z轴#1腔放料位触发标志
ANDNOT W363.04  ; 进料伺服Z轴取料位触发标志
ANDNOT W363.03  ; 进料伺服Z轴待机位触发标志
AND D1055.03  ; 进料伺服机构Z轴#1|2|3腔放料位4（步）
AND W211.04  ; #3氦检腔有放料需求标志
AND 850.06  ; 进料伺服X轴#3腔放料位标志
AND 803.08  ; #3腔体有料感应1标志[0003.08]
AND 803.09  ; #3腔体有料感应2标志[0003.09]
OUT W363.07  ; 进料伺服Z轴#3腔放料位触发标志
LD TR4
ANDNOT W363.07  ; 进料伺服Z轴#3腔放料位触发标志
ANDNOT W363.06  ; 进料伺服Z轴#2腔放料位触发标志
ANDNOT W363.05  ; 进料伺服Z轴#1腔放料位触发标志
ANDNOT W363.04  ; 进料伺服Z轴取料位触发标志
ANDNOT W363.03  ; 进料伺服Z轴待机位触发标志
AND D1055.03  ; 进料伺服机构Z轴#1|2|3腔放料位4（步）
AND W211.05  ; #4氦检腔有放料需求标志
AND 850.14  ; 进料伺服X轴#4腔放料位标志
AND 830.12  ; 4#腔体有料感应1标志[0030.12]
AND 830.13  ; 4#腔体有料感应2标志[0030.13]
OUT W363.12  ; 进料伺服Z轴#4腔放料位触发标志
LD TR3
ANDNOT W363.12  ; 进料伺服Z轴#4腔放料位触发标志
ANDNOT W363.07  ; 进料伺服Z轴#3腔放料位触发标志
ANDNOT W363.06  ; 进料伺服Z轴#2腔放料位触发标志
ANDNOT W363.05  ; 进料伺服Z轴#1腔放料位触发标志
ANDNOT W363.04  ; 进料伺服Z轴取料位触发标志
ANDNOT W363.03  ; 进料伺服Z轴待机位触发标志
AND D1049.02  ; 进料伺服机构Z轴#1|2夹爪扫码NG放料位2（步）
AND 850.07  ; 进料伺服X轴#1夹爪扫码NG放料位标志
AND H20.04  ; #1进料夹爪有NG料记忆
AND 800.08  ; #1进料夹爪夹紧位标志[0000.08]
OUT W363.08  ; 进料伺服Z轴#1夹爪扫码NG放料位触发标志
LD TR2
ANDNOT W363.08  ; 进料伺服Z轴#1夹爪扫码NG放料位触发标志
ANDNOT W363.12  ; 进料伺服Z轴#4腔放料位触发标志
ANDNOT W363.07  ; 进料伺服Z轴#3腔放料位触发标志
ANDNOT W363.06  ; 进料伺服Z轴#2腔放料位触发标志
ANDNOT W363.05  ; 进料伺服Z轴#1腔放料位触发标志
ANDNOT W363.04  ; 进料伺服Z轴取料位触发标志
ANDNOT W363.03  ; 进料伺服Z轴待机位触发标志
AND D1049.02  ; 进料伺服机构Z轴#1|2夹爪扫码NG放料位2（步）
AND 850.08  ; 进料伺服X轴#2夹爪扫码NG放料位标志
AND H20.06  ; #2进料夹爪有NG料记忆
ANDNOT H20.04  ; #1进料夹爪有NG料记忆
AND 800.10  ; #2进料夹爪夹紧位标志[0000.10]
OUT W363.09  ; 进料伺服Z轴#2夹爪扫码NG放料位触发标志
LD TR1
ANDNOT W363.09  ; 进料伺服Z轴#2夹爪扫码NG放料位触发标志
ANDNOT W363.08  ; 进料伺服Z轴#1夹爪扫码NG放料位触发标志
ANDNOT W363.12  ; 进料伺服Z轴#4腔放料位触发标志
ANDNOT W363.07  ; 进料伺服Z轴#3腔放料位触发标志
ANDNOT W363.06  ; 进料伺服Z轴#2腔放料位触发标志
ANDNOT W363.05  ; 进料伺服Z轴#1腔放料位触发标志
ANDNOT W363.04  ; 进料伺服Z轴取料位触发标志
ANDNOT W363.03  ; 进料伺服Z轴待机位触发标志
AND D1052.02  ; 进料伺服机构Z轴#1|2夹爪配对取放料位3（步）
LD W211.00  ; 进料伺服有配对放料需求标志
ANDNOT H20.02  ; 进料配对位有料记忆
ANDNOT 806.09  ; 进料配对位有料感应标志[0006.09]
AND H20.00  ; #1进料夹爪有料记忆
AND 800.08  ; #1进料夹爪夹紧位标志[0000.08]
AND H20.03  ; #1进料夹爪有OK料记忆
ANDNOT H20.01  ; #2进料夹爪有料记忆
LD W211.01  ; 进料伺服有配对取料需求标志
AND H20.02  ; 进料配对位有料记忆
AND 806.09  ; 进料配对位有料感应标志[0006.09]
LD H20.01  ; #2进料夹爪有料记忆
AND 800.10  ; #2进料夹爪夹紧位标志[0000.10]
AND H20.05  ; #2进料夹爪有OK料记忆
ANDNOT H20.00  ; #1进料夹爪有料记忆
LD W1.11  ; 清料时单个料有效选择
AND 200.05  ; 清料停止中
ANDNOT H10.00  ; #1扫码阻挡有料记忆
ANDNOT H10.01  ; #1进料位有料记忆
ANDNOT H12.00  ; #2扫码阻挡有料记忆
ANDNOT H12.01  ; #2进料位有料记忆
ANDNOT H20.00  ; #1进料夹爪有料记忆
ANDNOT H20.01  ; #2进料夹爪有料记忆
ORLD
ANDLD
AND 800.09  ; #1进料夹爪松开位标志[0000.09]
ORLD
ANDLD
AND 850.09  ; 进料伺服X轴#1夹爪配对取放料位标志
OUT W363.10  ; 进料伺服Z轴#1夹爪配对取放料位触发标志
LD TR0
ANDNOT W363.10  ; 进料伺服Z轴#1夹爪配对取放料位触发标志
ANDNOT W363.09  ; 进料伺服Z轴#2夹爪扫码NG放料位触发标志
ANDNOT W363.08  ; 进料伺服Z轴#1夹爪扫码NG放料位触发标志
ANDNOT W363.12  ; 进料伺服Z轴#4腔放料位触发标志
ANDNOT W363.07  ; 进料伺服Z轴#3腔放料位触发标志
ANDNOT W363.06  ; 进料伺服Z轴#2腔放料位触发标志
ANDNOT W363.05  ; 进料伺服Z轴#1腔放料位触发标志
ANDNOT W363.04  ; 进料伺服Z轴取料位触发标志
ANDNOT W363.03  ; 进料伺服Z轴待机位触发标志
AND D1052.02  ; 进料伺服机构Z轴#1|2夹爪配对取放料位3（步）
LD W211.00  ; 进料伺服有配对放料需求标志
ANDNOT H20.02  ; 进料配对位有料记忆
ANDNOT 806.09  ; 进料配对位有料感应标志[0006.09]
AND H20.01  ; #2进料夹爪有料记忆
AND 800.10  ; #2进料夹爪夹紧位标志[0000.10]
AND H20.05  ; #2进料夹爪有OK料记忆
ANDNOT H20.00  ; #1进料夹爪有料记忆
LD W211.01  ; 进料伺服有配对取料需求标志
AND H20.02  ; 进料配对位有料记忆
AND 806.09  ; 进料配对位有料感应标志[0006.09]
AND H20.00  ; #1进料夹爪有料记忆
AND 800.08  ; #1进料夹爪夹紧位标志[0000.08]
AND H20.03  ; #1进料夹爪有OK料记忆
ANDNOT H20.01  ; #2进料夹爪有料记忆
AND 800.11  ; #2进料夹爪松开位标志[0000.11]
ORLD
ANDLD
AND 850.10  ; 进料伺服X轴#2夹爪配对取放料位标志
OUT W363.11  ; 进料伺服Z轴#2夹爪配对取放料位触发标志

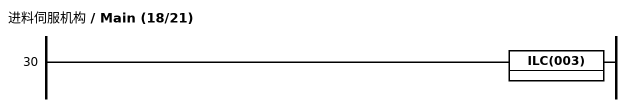
; rung 30
ILC(003)

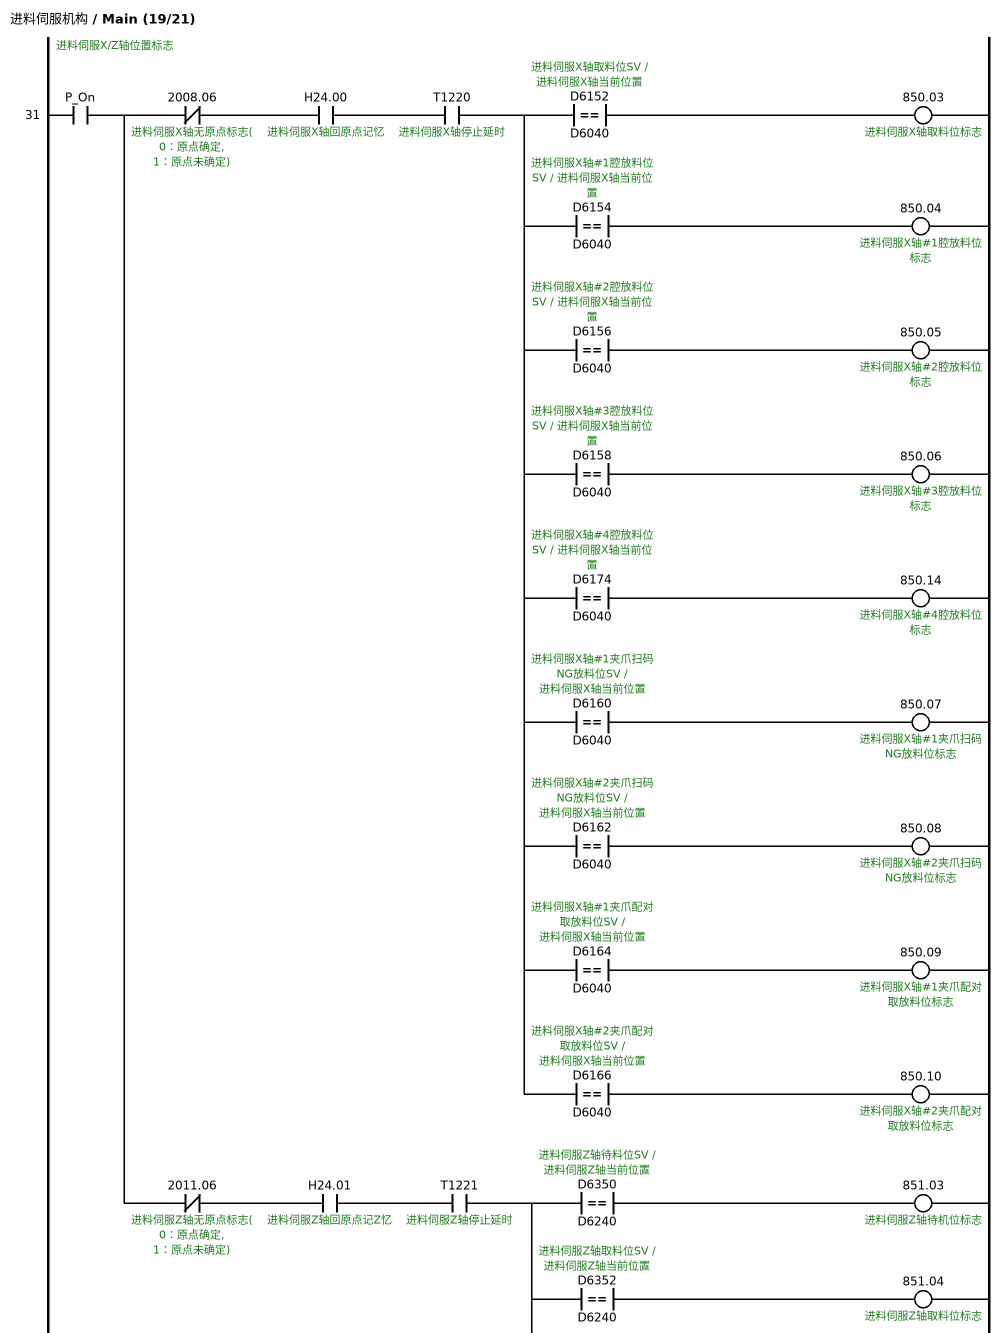

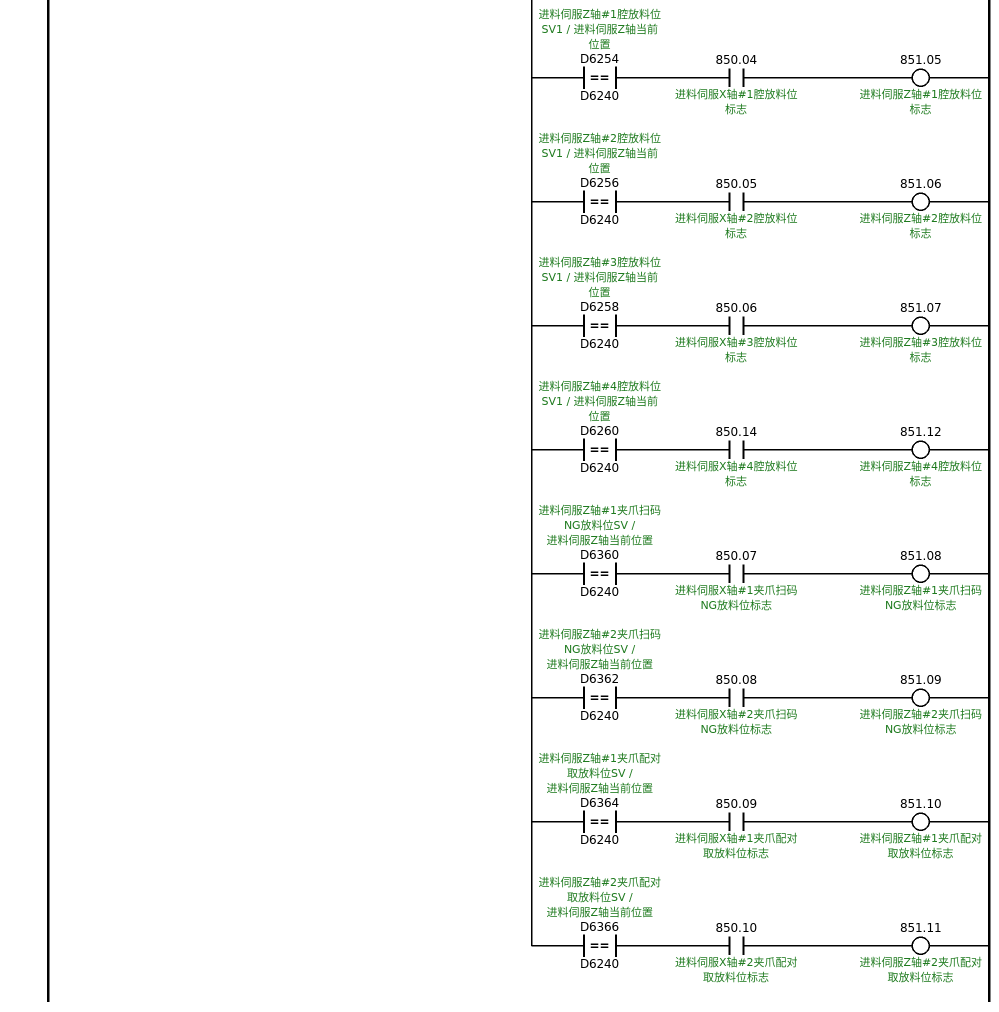
; rung 31: 进料伺服X/Z轴位置标志
LD P_On
OUT TR0
ANDNOT 2008.06  ; 进料伺服X轴无原点标志(0：原点确定,1：原点未确定)
AND H24.00  ; 进料伺服X轴回原点记忆
AND T1220  ; 进料伺服X轴停止延时
OUT TR1
AND=SL(303) D6152 D6040  ; 进料伺服X轴取料位SV, 进料伺服X轴当前位置
OUT 850.03  ; 进料伺服X轴取料位标志
LD TR1
AND=SL(303) D6154 D6040  ; 进料伺服X轴#1腔放料位SV, 进料伺服X轴当前位置
OUT 850.04  ; 进料伺服X轴#1腔放料位标志
LD TR1
AND=SL(303) D6156 D6040  ; 进料伺服X轴#2腔放料位SV, 进料伺服X轴当前位置
OUT 850.05  ; 进料伺服X轴#2腔放料位标志
LD TR1
AND=SL(303) D6158 D6040  ; 进料伺服X轴#3腔放料位SV, 进料伺服X轴当前位置
OUT 850.06  ; 进料伺服X轴#3腔放料位标志
LD TR1
AND=SL(303) D6174 D6040  ; 进料伺服X轴#4腔放料位SV, 进料伺服X轴当前位置
OUT 850.14  ; 进料伺服X轴#4腔放料位标志
LD TR1
AND=SL(303) D6160 D6040  ; 进料伺服X轴#1夹爪扫码NG放料位SV, 进料伺服X轴当前位置
OUT 850.07  ; 进料伺服X轴#1夹爪扫码NG放料位标志
LD TR1
AND=SL(303) D6162 D6040  ; 进料伺服X轴#2夹爪扫码NG放料位SV, 进料伺服X轴当前位置
OUT 850.08  ; 进料伺服X轴#2夹爪扫码NG放料位标志
LD TR1
AND=SL(303) D6164 D6040  ; 进料伺服X轴#1夹爪配对取放料位SV, 进料伺服X轴当前位置
OUT 850.09  ; 进料伺服X轴#1夹爪配对取放料位标志
LD TR1
AND=SL(303) D6166 D6040  ; 进料伺服X轴#2夹爪配对取放料位SV, 进料伺服X轴当前位置
OUT 850.10  ; 进料伺服X轴#2夹爪配对取放料位标志
LD TR0
ANDNOT 2011.06  ; 进料伺服Z轴无原点标志(0：原点确定,1：原点未确定)
AND H24.01  ; 进料伺服Z轴回原点记Z忆
AND T1221  ; 进料伺服Z轴停止延时
OUT TR0
AND=SL(303) D6350 D6240  ; 进料伺服Z轴待料位SV, 进料伺服Z轴当前位置
OUT 851.03  ; 进料伺服Z轴待机位标志
LD TR0
AND=SL(303) D6352 D6240  ; 进料伺服Z轴取料位SV, 进料伺服Z轴当前位置
OUT 851.04  ; 进料伺服Z轴取料位标志
LD TR0
AND=SL(303) D6254 D6240  ; 进料伺服Z轴#1腔放料位SV1, 进料伺服Z轴当前位置
AND 850.04  ; 进料伺服X轴#1腔放料位标志
OUT 851.05  ; 进料伺服Z轴#1腔放料位标志
LD TR0
AND=SL(303) D6256 D6240  ; 进料伺服Z轴#2腔放料位SV1, 进料伺服Z轴当前位置
AND 850.05  ; 进料伺服X轴#2腔放料位标志
OUT 851.06  ; 进料伺服Z轴#2腔放料位标志
LD TR0
AND=SL(303) D6258 D6240  ; 进料伺服Z轴#3腔放料位SV1, 进料伺服Z轴当前位置
AND 850.06  ; 进料伺服X轴#3腔放料位标志
OUT 851.07  ; 进料伺服Z轴#3腔放料位标志
LD TR0
AND=SL(303) D6260 D6240  ; 进料伺服Z轴#4腔放料位SV1, 进料伺服Z轴当前位置
AND 850.14  ; 进料伺服X轴#4腔放料位标志
OUT 851.12  ; 进料伺服Z轴#4腔放料位标志
LD TR0
AND=SL(303) D6360 D6240  ; 进料伺服Z轴#1夹爪扫码NG放料位SV, 进料伺服Z轴当前位置
AND 850.07  ; 进料伺服X轴#1夹爪扫码NG放料位标志
OUT 851.08  ; 进料伺服Z轴#1夹爪扫码NG放料位标志
LD TR0
AND=SL(303) D6362 D6240  ; 进料伺服Z轴#2夹爪扫码NG放料位SV, 进料伺服Z轴当前位置
AND 850.08  ; 进料伺服X轴#2夹爪扫码NG放料位标志
OUT 851.09  ; 进料伺服Z轴#2夹爪扫码NG放料位标志
LD TR0
AND=SL(303) D6364 D6240  ; 进料伺服Z轴#1夹爪配对取放料位SV, 进料伺服Z轴当前位置
AND 850.09  ; 进料伺服X轴#1夹爪配对取放料位标志
OUT 851.10  ; 进料伺服Z轴#1夹爪配对取放料位标志
LD TR0
AND=SL(303) D6366 D6240  ; 进料伺服Z轴#2夹爪配对取放料位SV, 进料伺服Z轴当前位置
AND 850.10  ; 进料伺服X轴#2夹爪配对取放料位标志
OUT 851.11  ; 进料伺服Z轴#2夹爪配对取放料位标志

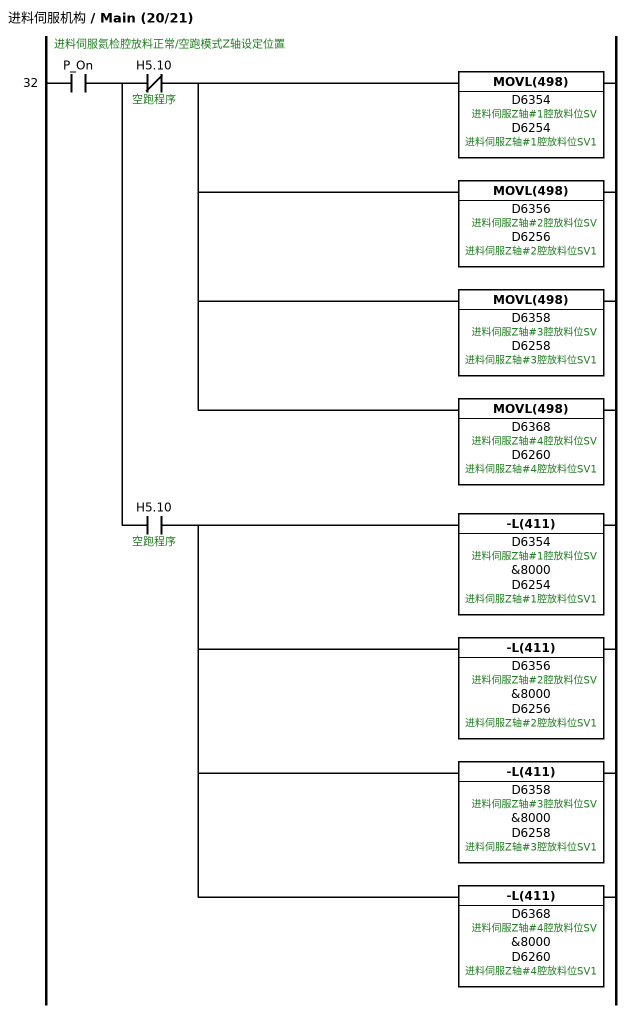
; rung 32: 进料伺服氦检腔放料正常/空跑模式Z轴设定位置
LD P_On
OUT TR0
ANDNOT H5.10  ; 空跑程序
MOVL(498) D6354 D6254  ; 进料伺服Z轴#1腔放料位SV, 进料伺服Z轴#1腔放料位SV1
MOVL(498) D6356 D6256  ; 进料伺服Z轴#2腔放料位SV, 进料伺服Z轴#2腔放料位SV1
MOVL(498) D6358 D6258  ; 进料伺服Z轴#3腔放料位SV, 进料伺服Z轴#3腔放料位SV1
MOVL(498) D6368 D6260  ; 进料伺服Z轴#4腔放料位SV, 进料伺服Z轴#4腔放料位SV1
LD TR0
AND H5.10  ; 空跑程序
-L(411) D6354 &8000 D6254  ; 进料伺服Z轴#1腔放料位SV, 进料伺服Z轴#1腔放料位SV1
-L(411) D6356 &8000 D6256  ; 进料伺服Z轴#2腔放料位SV, 进料伺服Z轴#2腔放料位SV1
-L(411) D6358 &8000 D6258  ; 进料伺服Z轴#3腔放料位SV, 进料伺服Z轴#3腔放料位SV1
-L(411) D6368 &8000 D6260  ; 进料伺服Z轴#4腔放料位SV, 进料伺服Z轴#4腔放料位SV1

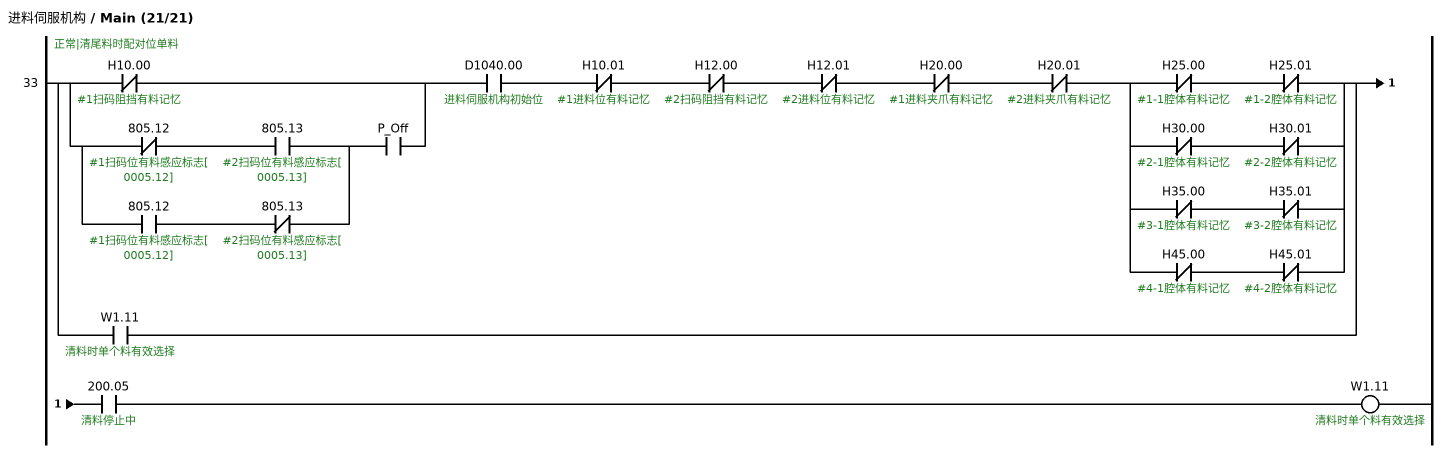
; rung 33: 正常|清尾料时配对位单料
LDNOT H10.00  ; #1扫码阻挡有料记忆
LDNOT 805.12  ; #1扫码位有料感应标志[0005.12]
AND 805.13  ; #2扫码位有料感应标志[0005.13]
LD 805.12  ; #1扫码位有料感应标志[0005.12]
ANDNOT 805.13  ; #2扫码位有料感应标志[0005.13]
ORLD
AND P_Off
ORLD
AND D1040.00  ; 进料伺服机构初始位
ANDNOT H10.01  ; #1进料位有料记忆
ANDNOT H12.00  ; #2扫码阻挡有料记忆
ANDNOT H12.01  ; #2进料位有料记忆
ANDNOT H20.00  ; #1进料夹爪有料记忆
ANDNOT H20.01  ; #2进料夹爪有料记忆
LDNOT H25.00  ; #1-1腔体有料记忆
ANDNOT H25.01  ; #1-2腔体有料记忆
LDNOT H30.00  ; #2-1腔体有料记忆
ANDNOT H30.01  ; #2-2腔体有料记忆
ORLD
LDNOT H35.00  ; #3-1腔体有料记忆
ANDNOT H35.01  ; #3-2腔体有料记忆
ORLD
LDNOT H45.00  ; #4-1腔体有料记忆
ANDNOT H45.01  ; #4-2腔体有料记忆
ORLD
ANDLD
OR W1.11  ; 清料时单个料有效选择
AND 200.05  ; 清料停止中
OUT W1.11  ; 清料时单个料有效选择

### Section 进料伺服手动

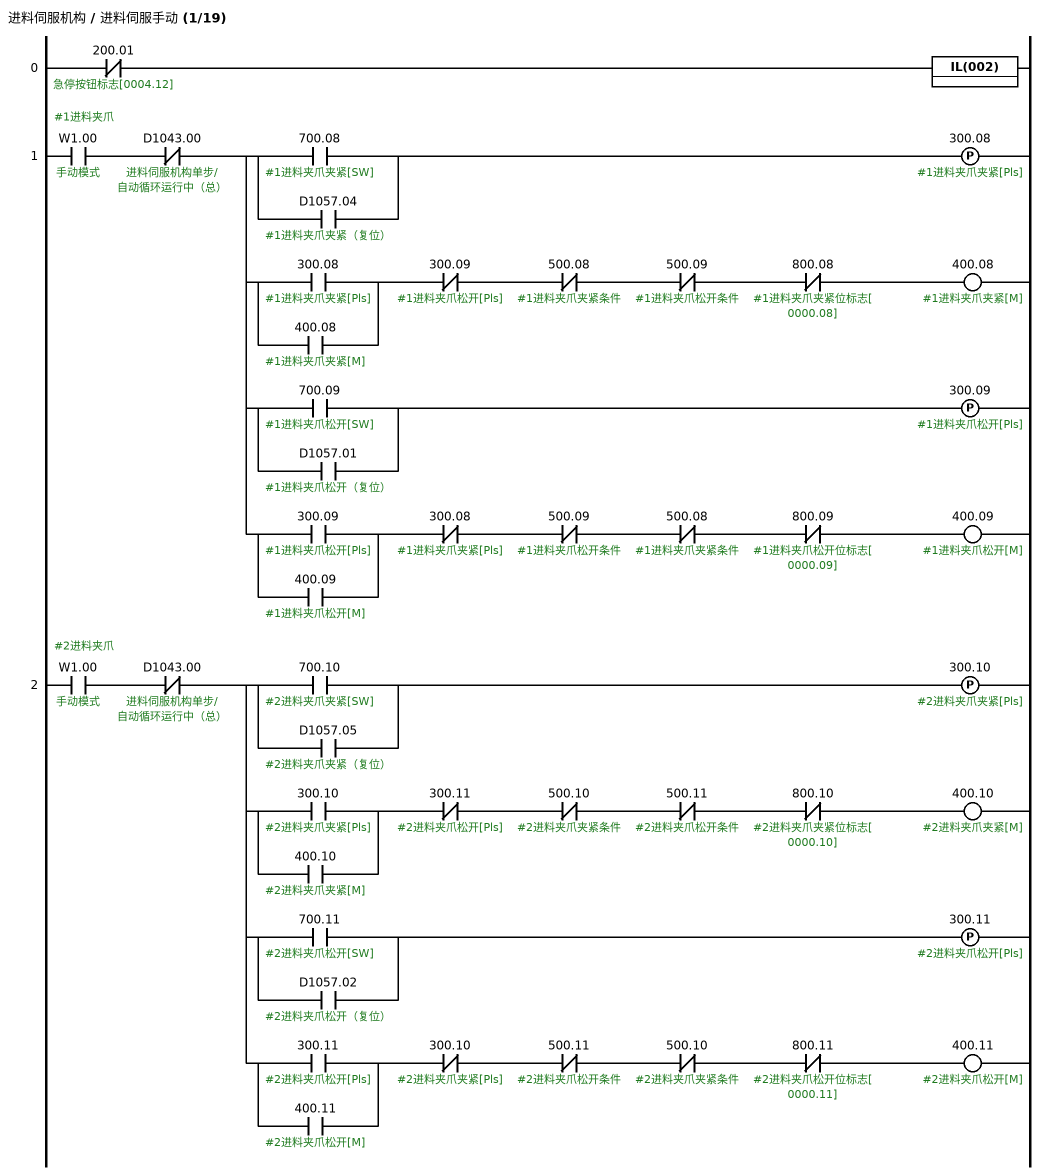
; rung 0
LDNOT 200.01  ; 急停按钮标志[0004.12]
IL(002)
; rung 1: #1进料夹爪
LD W1.00  ; 手动模式
ANDNOT D1043.00  ; 进料伺服机构单步/自动循环运行中（总）
OUT TR0
LD 700.08  ; #1进料夹爪夹紧[SW]
OR D1057.04  ; #1进料夹爪夹紧（复位）
ANDLD
DIFU(013) 300.08  ; #1进料夹爪夹紧[Pls]
LD TR0
LD 300.08  ; #1进料夹爪夹紧[Pls]
OR 400.08  ; #1进料夹爪夹紧[M]
ANDLD
ANDNOT 300.09  ; #1进料夹爪松开[Pls]
ANDNOT 500.08  ; #1进料夹爪夹紧条件
ANDNOT 500.09  ; #1进料夹爪松开条件
ANDNOT 800.08  ; #1进料夹爪夹紧位标志[0000.08]
OUT 400.08  ; #1进料夹爪夹紧[M]
LD TR0
LD 700.09  ; #1进料夹爪松开[SW]
OR D1057.01  ; #1进料夹爪松开（复位）
ANDLD
DIFU(013) 300.09  ; #1进料夹爪松开[Pls]
LD TR0
LD 300.09  ; #1进料夹爪松开[Pls]
OR 400.09  ; #1进料夹爪松开[M]
ANDLD
ANDNOT 300.08  ; #1进料夹爪夹紧[Pls]
ANDNOT 500.09  ; #1进料夹爪松开条件
ANDNOT 500.08  ; #1进料夹爪夹紧条件
ANDNOT 800.09  ; #1进料夹爪松开位标志[0000.09]
OUT 400.09  ; #1进料夹爪松开[M]
; rung 2: #2进料夹爪
LD W1.00  ; 手动模式
ANDNOT D1043.00  ; 进料伺服机构单步/自动循环运行中（总）
OUT TR0
LD 700.10  ; #2进料夹爪夹紧[SW]
OR D1057.05  ; #2进料夹爪夹紧（复位）
ANDLD
DIFU(013) 300.10  ; #2进料夹爪夹紧[Pls]
LD TR0
LD 300.10  ; #2进料夹爪夹紧[Pls]
OR 400.10  ; #2进料夹爪夹紧[M]
ANDLD
ANDNOT 300.11  ; #2进料夹爪松开[Pls]
ANDNOT 500.10  ; #2进料夹爪夹紧条件
ANDNOT 500.11  ; #2进料夹爪松开条件
ANDNOT 800.10  ; #2进料夹爪夹紧位标志[0000.10]
OUT 400.10  ; #2进料夹爪夹紧[M]
LD TR0
LD 700.11  ; #2进料夹爪松开[SW]
OR D1057.02  ; #2进料夹爪松开（复位）
ANDLD
DIFU(013) 300.11  ; #2进料夹爪松开[Pls]
LD TR0
LD 300.11  ; #2进料夹爪松开[Pls]
OR 400.11  ; #2进料夹爪松开[M]
ANDLD
ANDNOT 300.10  ; #2进料夹爪夹紧[Pls]
ANDNOT 500.11  ; #2进料夹爪松开条件
ANDNOT 500.10  ; #2进料夹爪夹紧条件
ANDNOT 800.11  ; #2进料夹爪松开位标志[0000.11]
OUT 400.11  ; #2进料夹爪松开[M]

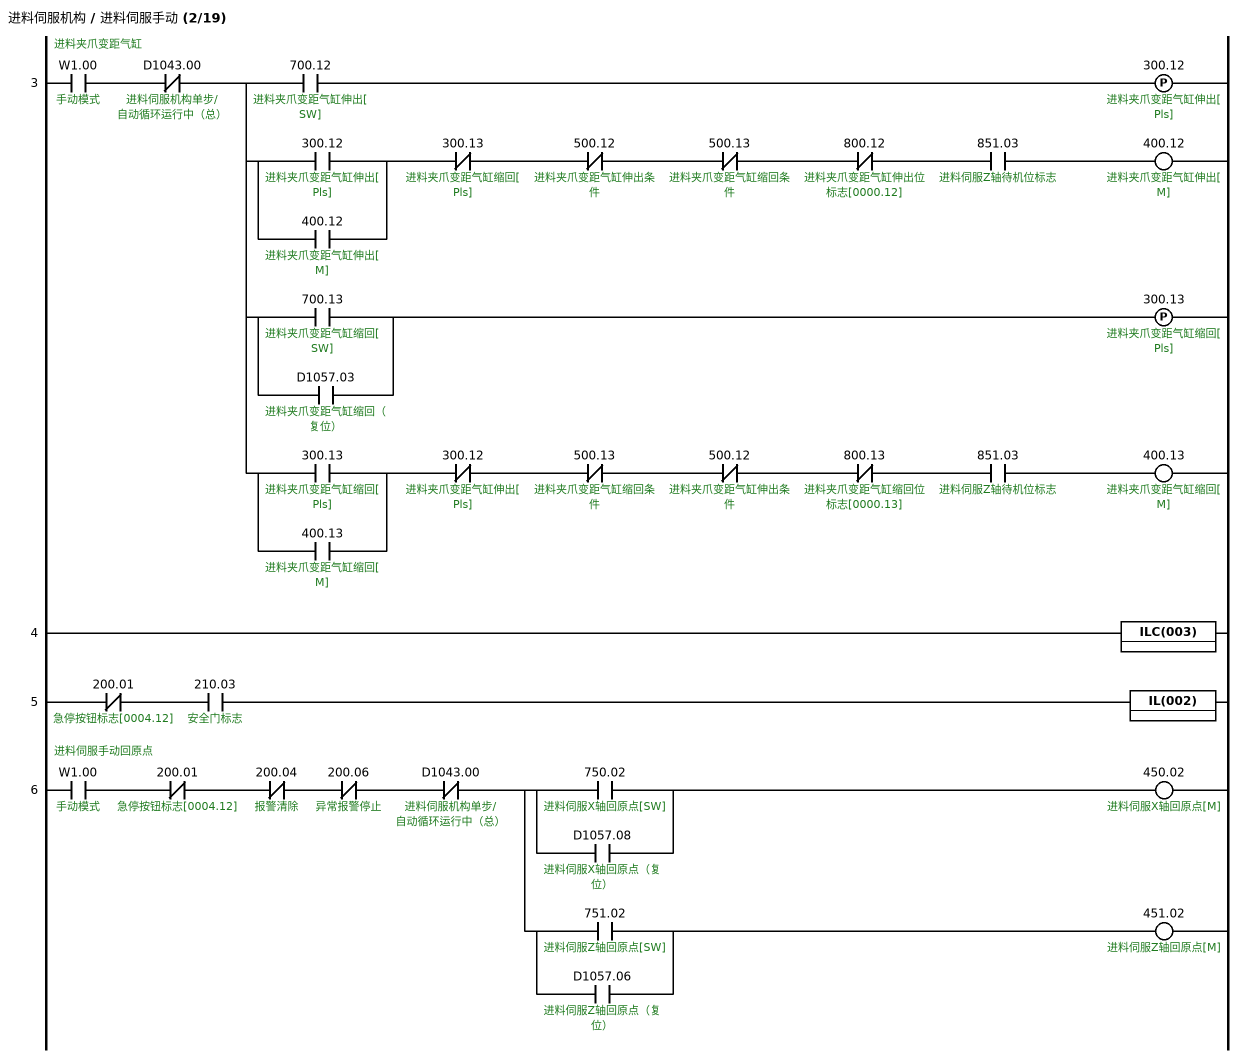
; rung 3: 进料夹爪变距气缸
LD W1.00  ; 手动模式
ANDNOT D1043.00  ; 进料伺服机构单步/自动循环运行中（总）
OUT TR0
AND 700.12  ; 进料夹爪变距气缸伸出[SW]
DIFU(013) 300.12  ; 进料夹爪变距气缸伸出[Pls]
LD TR0
LD 300.12  ; 进料夹爪变距气缸伸出[Pls]
OR 400.12  ; 进料夹爪变距气缸伸出[M]
ANDLD
ANDNOT 300.13  ; 进料夹爪变距气缸缩回[Pls]
ANDNOT 500.12  ; 进料夹爪变距气缸伸出条件
ANDNOT 500.13  ; 进料夹爪变距气缸缩回条件
ANDNOT 800.12  ; 进料夹爪变距气缸伸出位标志[0000.12]
AND 851.03  ; 进料伺服Z轴待机位标志
OUT 400.12  ; 进料夹爪变距气缸伸出[M]
LD TR0
LD 700.13  ; 进料夹爪变距气缸缩回[SW]
OR D1057.03  ; 进料夹爪变距气缸缩回（复位）
ANDLD
DIFU(013) 300.13  ; 进料夹爪变距气缸缩回[Pls]
LD TR0
LD 300.13  ; 进料夹爪变距气缸缩回[Pls]
OR 400.13  ; 进料夹爪变距气缸缩回[M]
ANDLD
ANDNOT 300.12  ; 进料夹爪变距气缸伸出[Pls]
ANDNOT 500.13  ; 进料夹爪变距气缸缩回条件
ANDNOT 500.12  ; 进料夹爪变距气缸伸出条件
ANDNOT 800.13  ; 进料夹爪变距气缸缩回位标志[0000.13]
AND 851.03  ; 进料伺服Z轴待机位标志
OUT 400.13  ; 进料夹爪变距气缸缩回[M]
; rung 4
ILC(003)
; rung 5
LDNOT 200.01  ; 急停按钮标志[0004.12]
AND 210.03  ; 安全门标志
IL(002)
; rung 6: 进料伺服手动回原点
LD W1.00  ; 手动模式
ANDNOT 200.01  ; 急停按钮标志[0004.12]
ANDNOT 200.04  ; 报警清除
ANDNOT 200.06  ; 异常报警停止
ANDNOT D1043.00  ; 进料伺服机构单步/自动循环运行中（总）
OUT TR0
LD 750.02  ; 进料伺服X轴回原点[SW]
OR D1057.08  ; 进料伺服X轴回原点（复位）
ANDLD
OUT 450.02  ; 进料伺服X轴回原点[M]
LD TR0
LD 751.02  ; 进料伺服Z轴回原点[SW]
OR D1057.06  ; 进料伺服Z轴回原点（复位）
ANDLD
OUT 451.02  ; 进料伺服Z轴回原点[M]

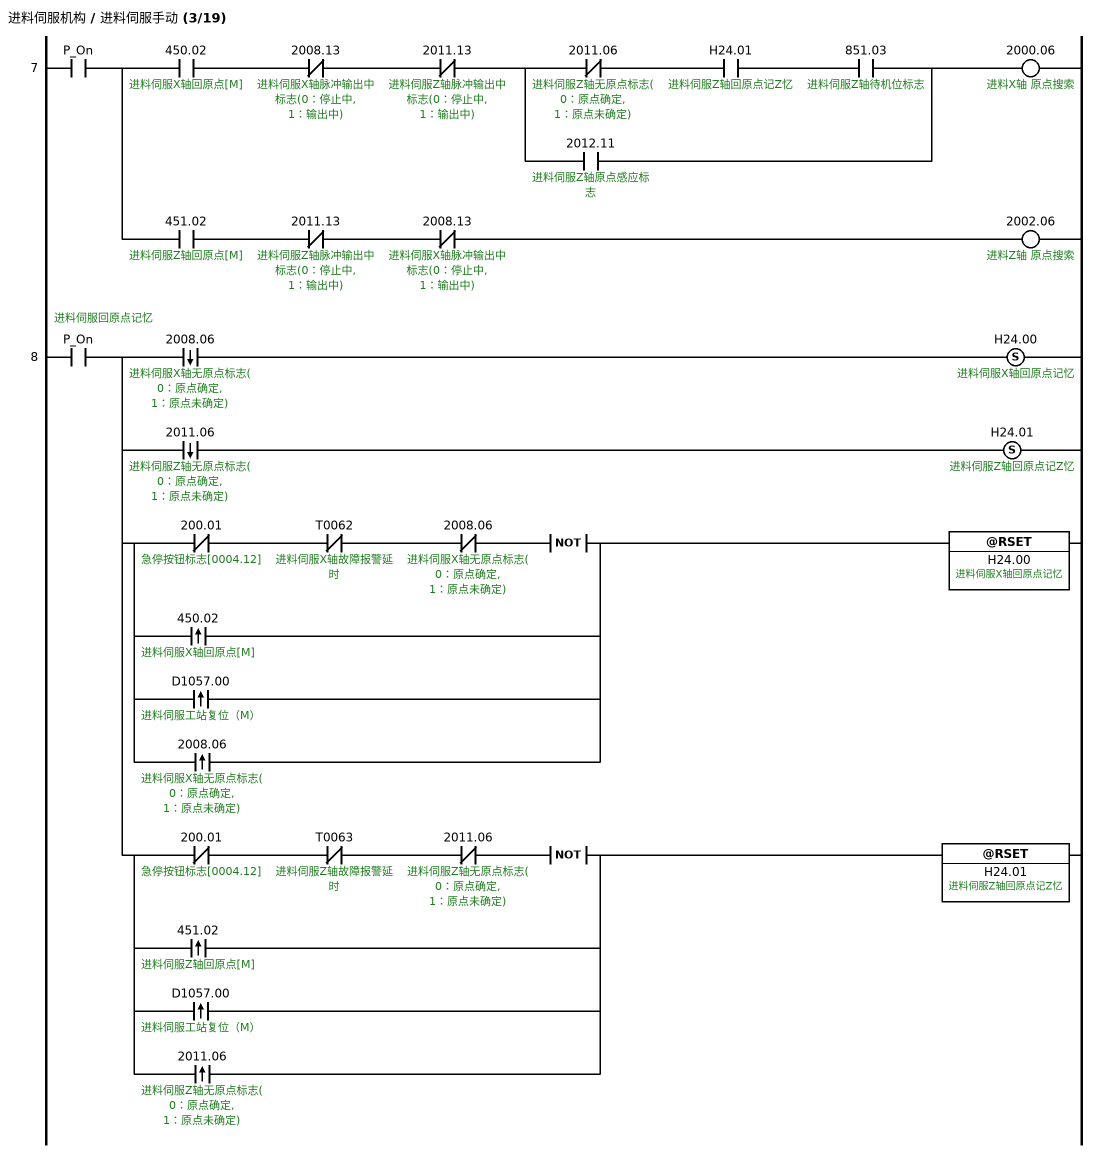
; rung 7
LD P_On
OUT TR0
AND 450.02  ; 进料伺服X轴回原点[M]
ANDNOT 2008.13  ; 进料伺服X轴脉冲输出中标志(0：停止中,1：输出中)
ANDNOT 2011.13  ; 进料伺服Z轴脉冲输出中标志(0：停止中,1：输出中)
LDNOT 2011.06  ; 进料伺服Z轴无原点标志(0：原点确定,1：原点未确定)
AND H24.01  ; 进料伺服Z轴回原点记Z忆
AND 851.03  ; 进料伺服Z轴待机位标志
OR 2012.11  ; 进料伺服Z轴原点感应标志
ANDLD
OUT 2000.06  ; 进料X轴 原点搜索
LD TR0
AND 451.02  ; 进料伺服Z轴回原点[M]
ANDNOT 2011.13  ; 进料伺服Z轴脉冲输出中标志(0：停止中,1：输出中)
ANDNOT 2008.13  ; 进料伺服X轴脉冲输出中标志(0：停止中,1：输出中)
OUT 2002.06  ; 进料Z轴 原点搜索
; rung 8: 进料伺服回原点记忆
LD P_On
OUT TR0
%AND 2008.06  ; 进料伺服X轴无原点标志(0：原点确定,1：原点未确定)
SET H24.00  ; 进料伺服X轴回原点记忆
LD TR0
%AND 2011.06  ; 进料伺服Z轴无原点标志(0：原点确定,1：原点未确定)
SET H24.01  ; 进料伺服Z轴回原点记Z忆
LD TR0
LDNOT 200.01  ; 急停按钮标志[0004.12]
ANDNOT T0062  ; 进料伺服X轴故障报警延时
ANDNOT 2008.06  ; 进料伺服X轴无原点标志(0：原点确定,1：原点未确定)
NOT(520)
@OR 450.02  ; 进料伺服X轴回原点[M]
@OR D1057.00  ; 进料伺服工站复位（M）
@OR 2008.06  ; 进料伺服X轴无原点标志(0：原点确定,1：原点未确定)
ANDLD
@RSET H24.00  ; 进料伺服X轴回原点记忆
LD TR0
LDNOT 200.01  ; 急停按钮标志[0004.12]
ANDNOT T0063  ; 进料伺服Z轴故障报警延时
ANDNOT 2011.06  ; 进料伺服Z轴无原点标志(0：原点确定,1：原点未确定)
NOT(520)
@OR 451.02  ; 进料伺服Z轴回原点[M]
@OR D1057.00  ; 进料伺服工站复位（M）
@OR 2011.06  ; 进料伺服Z轴无原点标志(0：原点确定,1：原点未确定)
ANDLD
@RSET H24.01  ; 进料伺服Z轴回原点记Z忆

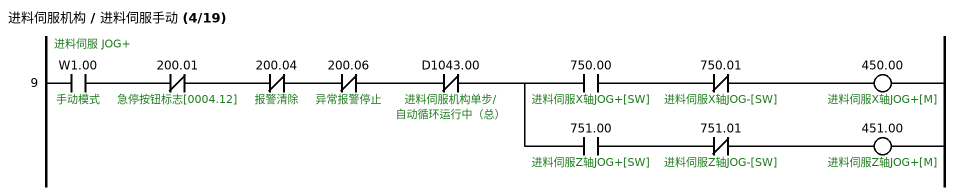
; rung 9: 进料伺服 JOG+
LD W1.00  ; 手动模式
ANDNOT 200.01  ; 急停按钮标志[0004.12]
ANDNOT 200.04  ; 报警清除
ANDNOT 200.06  ; 异常报警停止
ANDNOT D1043.00  ; 进料伺服机构单步/自动循环运行中（总）
OUT TR0
AND 750.00  ; 进料伺服X轴JOG+[SW]
ANDNOT 750.01  ; 进料伺服X轴JOG-[SW]
OUT 450.00  ; 进料伺服X轴JOG+[M]
LD TR0
AND 751.00  ; 进料伺服Z轴JOG+[SW]
ANDNOT 751.01  ; 进料伺服Z轴JOG-[SW]
OUT 451.00  ; 进料伺服Z轴JOG+[M]

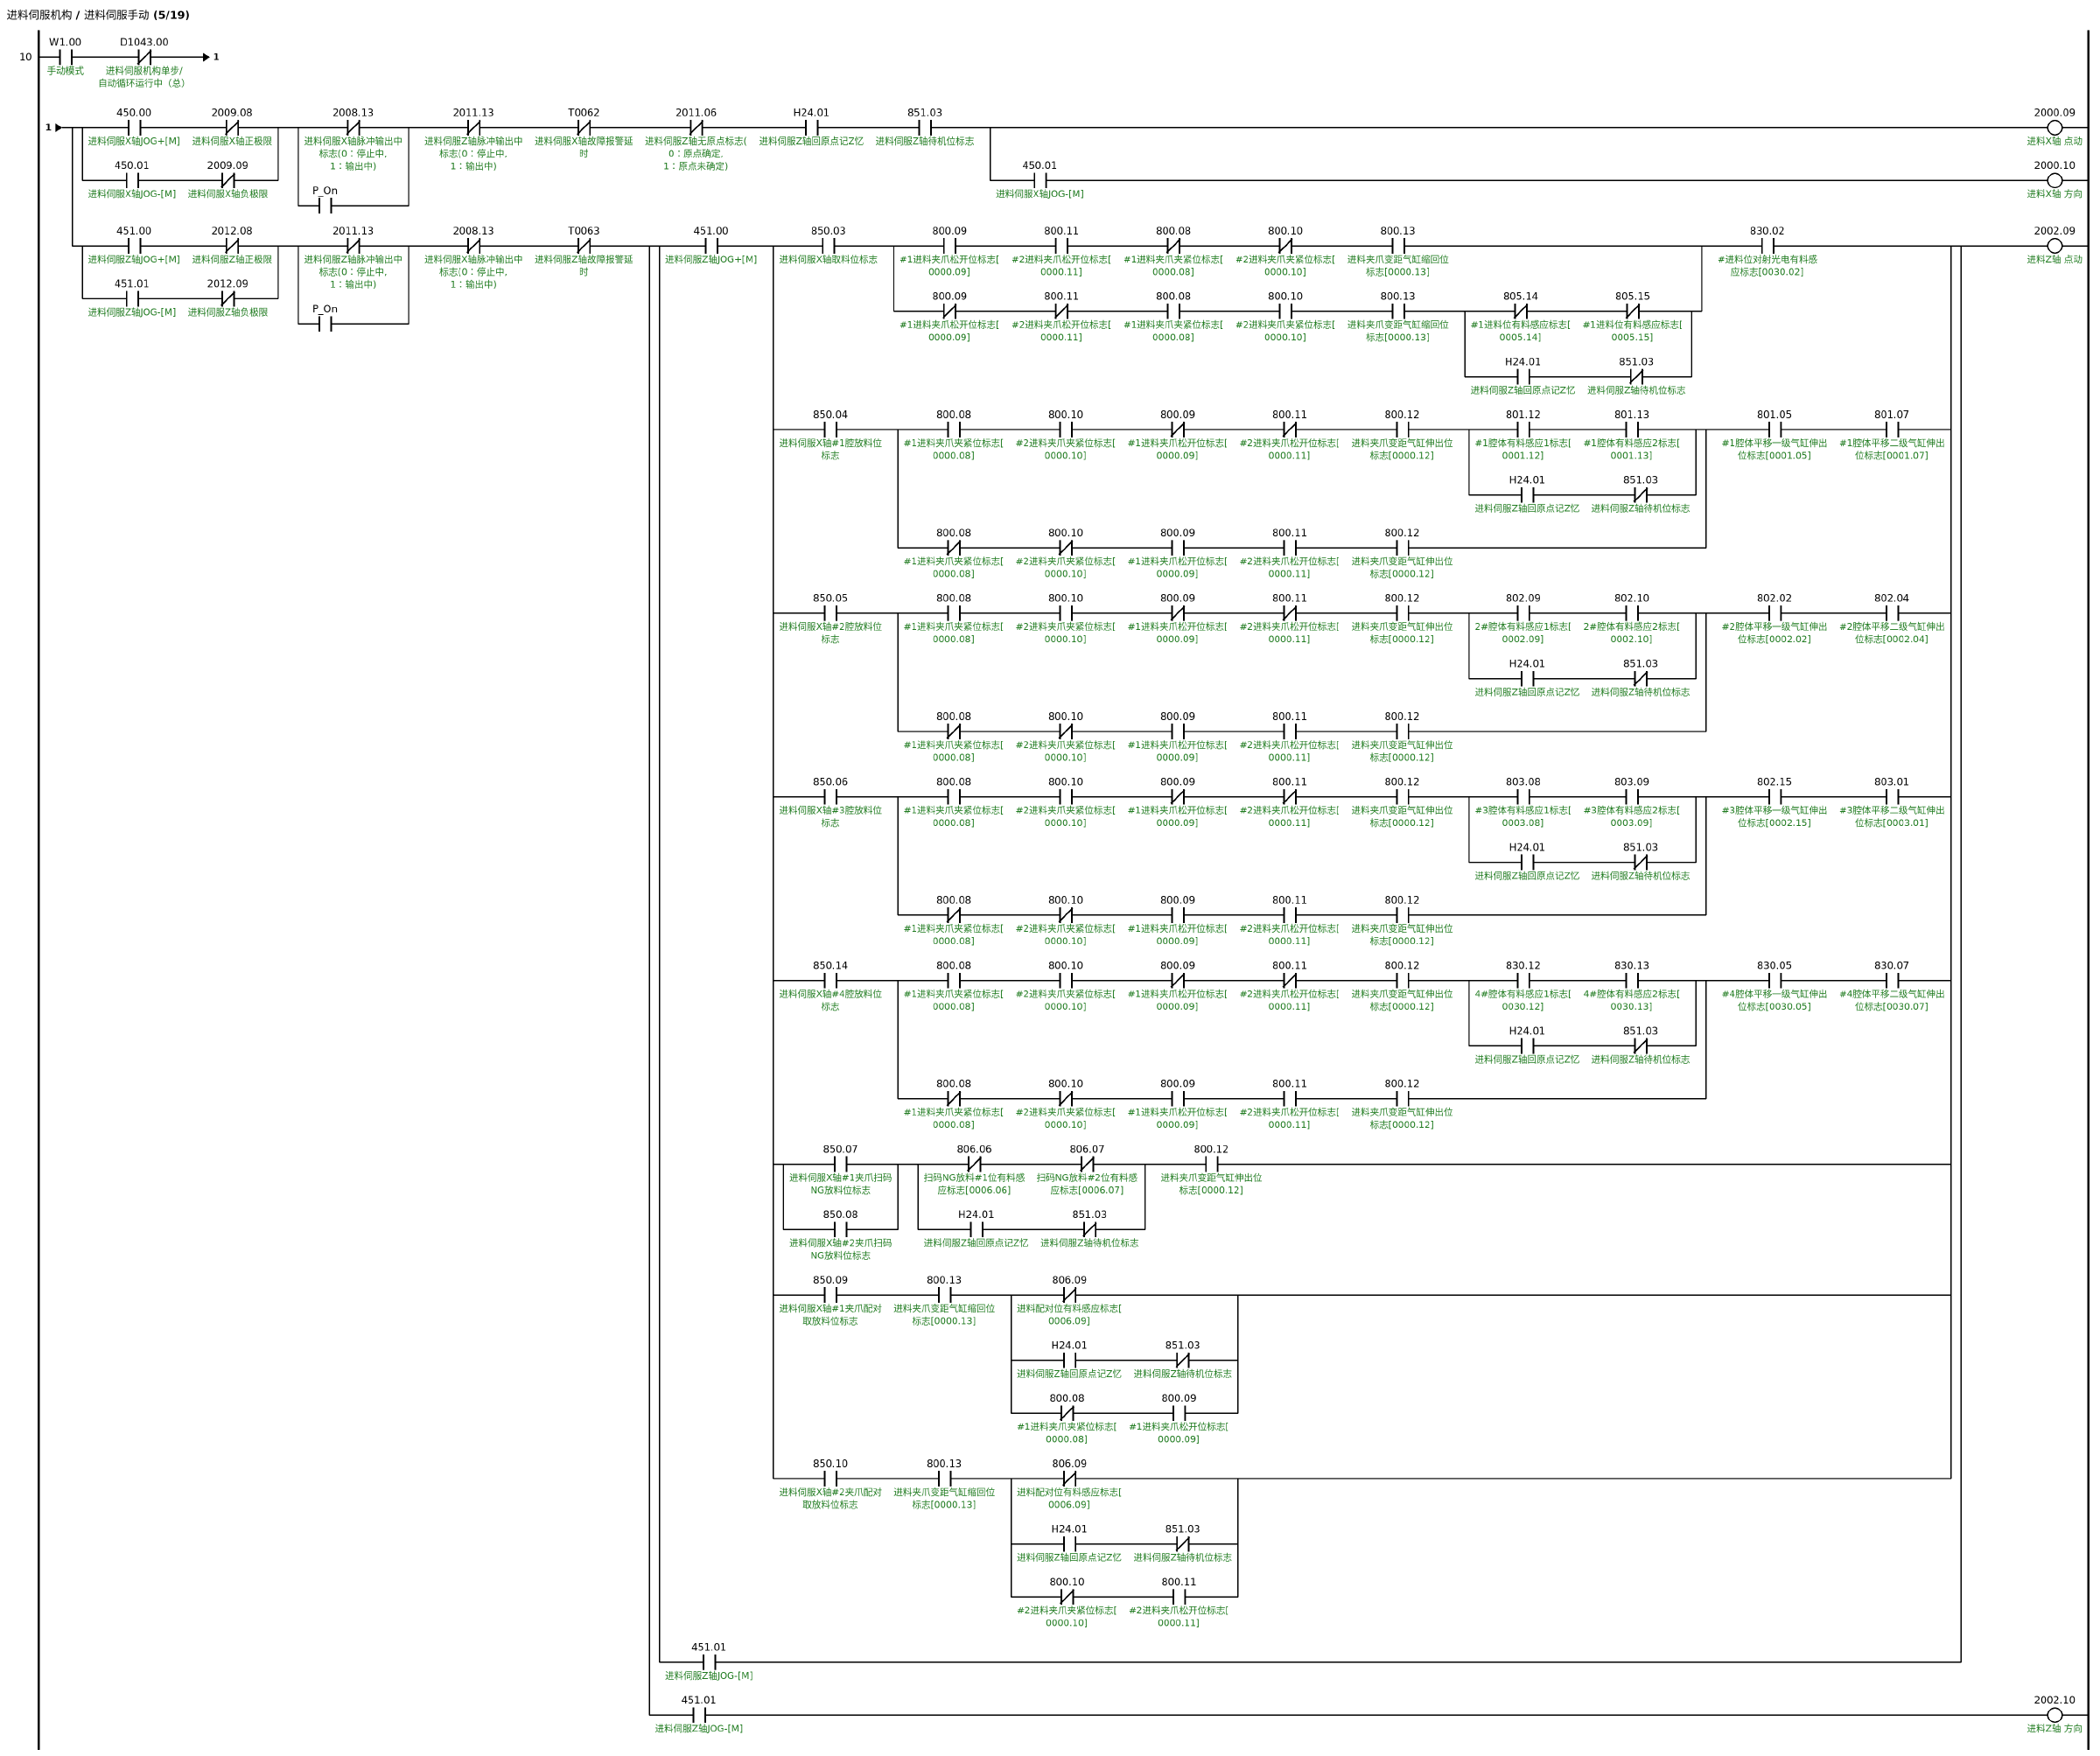
; rung 10
LD W1.00  ; 手动模式
ANDNOT D1043.00  ; 进料伺服机构单步/自动循环运行中（总）
OUT TR0
LD 450.00  ; 进料伺服X轴JOG+[M]
ANDNOT 2009.08  ; 进料伺服X轴正极限
LD 450.01  ; 进料伺服X轴JOG-[M]
ANDNOT 2009.09  ; 进料伺服X轴负极限
ORLD
ANDLD
LDNOT 2008.13  ; 进料伺服X轴脉冲输出中标志(0：停止中,1：输出中)
OR P_On
ANDLD
ANDNOT 2011.13  ; 进料伺服Z轴脉冲输出中标志(0：停止中,1：输出中)
ANDNOT T0062  ; 进料伺服X轴故障报警延时
ANDNOT 2011.06  ; 进料伺服Z轴无原点标志(0：原点确定,1：原点未确定)
AND H24.01  ; 进料伺服Z轴回原点记Z忆
AND 851.03  ; 进料伺服Z轴待机位标志
OUT 2000.09  ; 进料X轴 点动
AND 450.01  ; 进料伺服X轴JOG-[M]
OUT 2000.10  ; 进料X轴 方向
LD TR0
LD 451.00  ; 进料伺服Z轴JOG+[M]
ANDNOT 2012.08  ; 进料伺服Z轴正极限
LD 451.01  ; 进料伺服Z轴JOG-[M]
ANDNOT 2012.09  ; 进料伺服Z轴负极限
ORLD
ANDLD
LDNOT 2011.13  ; 进料伺服Z轴脉冲输出中标志(0：停止中,1：输出中)
OR P_On
ANDLD
ANDNOT 2008.13  ; 进料伺服X轴脉冲输出中标志(0：停止中,1：输出中)
ANDNOT T0063  ; 进料伺服Z轴故障报警延时
OUT TR0
LD 451.00  ; 进料伺服Z轴JOG+[M]
LD 850.03  ; 进料伺服X轴取料位标志
LD 800.09  ; #1进料夹爪松开位标志[0000.09]
AND 800.11  ; #2进料夹爪松开位标志[0000.11]
ANDNOT 800.08  ; #1进料夹爪夹紧位标志[0000.08]
ANDNOT 800.10  ; #2进料夹爪夹紧位标志[0000.10]
AND 800.13  ; 进料夹爪变距气缸缩回位标志[0000.13]
LDNOT 800.09  ; #1进料夹爪松开位标志[0000.09]
ANDNOT 800.11  ; #2进料夹爪松开位标志[0000.11]
AND 800.08  ; #1进料夹爪夹紧位标志[0000.08]
AND 800.10  ; #2进料夹爪夹紧位标志[0000.10]
AND 800.13  ; 进料夹爪变距气缸缩回位标志[0000.13]
LDNOT 805.14  ; #1进料位有料感应标志[0005.14]
ANDNOT 805.15  ; #1进料位有料感应标志[0005.15]
LD H24.01  ; 进料伺服Z轴回原点记Z忆
ANDNOT 851.03  ; 进料伺服Z轴待机位标志
ORLD
ANDLD
ORLD
ANDLD
AND 830.02  ; #进料位对射光电有料感应标志[0030.02]
LD 850.04  ; 进料伺服X轴#1腔放料位标志
LD 800.08  ; #1进料夹爪夹紧位标志[0000.08]
AND 800.10  ; #2进料夹爪夹紧位标志[0000.10]
ANDNOT 800.09  ; #1进料夹爪松开位标志[0000.09]
ANDNOT 800.11  ; #2进料夹爪松开位标志[0000.11]
AND 800.12  ; 进料夹爪变距气缸伸出位标志[0000.12]
LD 801.12  ; #1腔体有料感应1标志[0001.12]
AND 801.13  ; #1腔体有料感应2标志[0001.13]
LD H24.01  ; 进料伺服Z轴回原点记Z忆
ANDNOT 851.03  ; 进料伺服Z轴待机位标志
ORLD
ANDLD
LDNOT 800.08  ; #1进料夹爪夹紧位标志[0000.08]
ANDNOT 800.10  ; #2进料夹爪夹紧位标志[0000.10]
AND 800.09  ; #1进料夹爪松开位标志[0000.09]
AND 800.11  ; #2进料夹爪松开位标志[0000.11]
AND 800.12  ; 进料夹爪变距气缸伸出位标志[0000.12]
ORLD
ANDLD
AND 801.05  ; #1腔体平移一级气缸伸出位标志[0001.05]
AND 801.07  ; #1腔体平移二级气缸伸出位标志[0001.07]
ORLD
LD 850.05  ; 进料伺服X轴#2腔放料位标志
LD 800.08  ; #1进料夹爪夹紧位标志[0000.08]
AND 800.10  ; #2进料夹爪夹紧位标志[0000.10]
ANDNOT 800.09  ; #1进料夹爪松开位标志[0000.09]
ANDNOT 800.11  ; #2进料夹爪松开位标志[0000.11]
AND 800.12  ; 进料夹爪变距气缸伸出位标志[0000.12]
LD 802.09  ; 2#腔体有料感应1标志[0002.09]
AND 802.10  ; 2#腔体有料感应2标志[0002.10]
LD H24.01  ; 进料伺服Z轴回原点记Z忆
ANDNOT 851.03  ; 进料伺服Z轴待机位标志
ORLD
ANDLD
LDNOT 800.08  ; #1进料夹爪夹紧位标志[0000.08]
ANDNOT 800.10  ; #2进料夹爪夹紧位标志[0000.10]
AND 800.09  ; #1进料夹爪松开位标志[0000.09]
AND 800.11  ; #2进料夹爪松开位标志[0000.11]
AND 800.12  ; 进料夹爪变距气缸伸出位标志[0000.12]
ORLD
ANDLD
AND 802.02  ; #2腔体平移一级气缸伸出位标志[0002.02]
AND 802.04  ; #2腔体平移二级气缸伸出位标志[0002.04]
ORLD
LD 850.06  ; 进料伺服X轴#3腔放料位标志
LD 800.08  ; #1进料夹爪夹紧位标志[0000.08]
AND 800.10  ; #2进料夹爪夹紧位标志[0000.10]
ANDNOT 800.09  ; #1进料夹爪松开位标志[0000.09]
ANDNOT 800.11  ; #2进料夹爪松开位标志[0000.11]
AND 800.12  ; 进料夹爪变距气缸伸出位标志[0000.12]
LD 803.08  ; #3腔体有料感应1标志[0003.08]
AND 803.09  ; #3腔体有料感应2标志[0003.09]
LD H24.01  ; 进料伺服Z轴回原点记Z忆
ANDNOT 851.03  ; 进料伺服Z轴待机位标志
ORLD
ANDLD
LDNOT 800.08  ; #1进料夹爪夹紧位标志[0000.08]
ANDNOT 800.10  ; #2进料夹爪夹紧位标志[0000.10]
AND 800.09  ; #1进料夹爪松开位标志[0000.09]
AND 800.11  ; #2进料夹爪松开位标志[0000.11]
AND 800.12  ; 进料夹爪变距气缸伸出位标志[0000.12]
ORLD
ANDLD
AND 802.15  ; #3腔体平移一级气缸伸出位标志[0002.15]
AND 803.01  ; #3腔体平移二级气缸伸出位标志[0003.01]
ORLD
LD 850.14  ; 进料伺服X轴#4腔放料位标志
LD 800.08  ; #1进料夹爪夹紧位标志[0000.08]
AND 800.10  ; #2进料夹爪夹紧位标志[0000.10]
ANDNOT 800.09  ; #1进料夹爪松开位标志[0000.09]
ANDNOT 800.11  ; #2进料夹爪松开位标志[0000.11]
AND 800.12  ; 进料夹爪变距气缸伸出位标志[0000.12]
LD 830.12  ; 4#腔体有料感应1标志[0030.12]
AND 830.13  ; 4#腔体有料感应2标志[0030.13]
LD H24.01  ; 进料伺服Z轴回原点记Z忆
ANDNOT 851.03  ; 进料伺服Z轴待机位标志
ORLD
ANDLD
LDNOT 800.08  ; #1进料夹爪夹紧位标志[0000.08]
ANDNOT 800.10  ; #2进料夹爪夹紧位标志[0000.10]
AND 800.09  ; #1进料夹爪松开位标志[0000.09]
AND 800.11  ; #2进料夹爪松开位标志[0000.11]
AND 800.12  ; 进料夹爪变距气缸伸出位标志[0000.12]
ORLD
ANDLD
AND 830.05  ; #4腔体平移一级气缸伸出位标志[0030.05]
AND 830.07  ; #4腔体平移二级气缸伸出位标志[0030.07]
ORLD
LD 850.07  ; 进料伺服X轴#1夹爪扫码NG放料位标志
OR 850.08  ; 进料伺服X轴#2夹爪扫码NG放料位标志
LDNOT 806.06  ; 扫码NG放料#1位有料感应标志[0006.06]
ANDNOT 806.07  ; 扫码NG放料#2位有料感应标志[0006.07]
LD H24.01  ; 进料伺服Z轴回原点记Z忆
ANDNOT 851.03  ; 进料伺服Z轴待机位标志
ORLD
ANDLD
AND 800.12  ; 进料夹爪变距气缸伸出位标志[0000.12]
ORLD
LD 850.09  ; 进料伺服X轴#1夹爪配对取放料位标志
AND 800.13  ; 进料夹爪变距气缸缩回位标志[0000.13]
LDNOT 806.09  ; 进料配对位有料感应标志[0006.09]
LD H24.01  ; 进料伺服Z轴回原点记Z忆
ANDNOT 851.03  ; 进料伺服Z轴待机位标志
ORLD
LDNOT 800.08  ; #1进料夹爪夹紧位标志[0000.08]
AND 800.09  ; #1进料夹爪松开位标志[0000.09]
ORLD
ANDLD
ORLD
LD 850.10  ; 进料伺服X轴#2夹爪配对取放料位标志
AND 800.13  ; 进料夹爪变距气缸缩回位标志[0000.13]
LDNOT 806.09  ; 进料配对位有料感应标志[0006.09]
LD H24.01  ; 进料伺服Z轴回原点记Z忆
ANDNOT 851.03  ; 进料伺服Z轴待机位标志
ORLD
LDNOT 800.10  ; #2进料夹爪夹紧位标志[0000.10]
AND 800.11  ; #2进料夹爪松开位标志[0000.11]
ORLD
ANDLD
ORLD
ANDLD
OR 451.01  ; 进料伺服Z轴JOG-[M]
ANDLD
OUT 2002.09  ; 进料Z轴 点动
LD TR0
AND 451.01  ; 进料伺服Z轴JOG-[M]
OUT 2002.10  ; 进料Z轴 方向

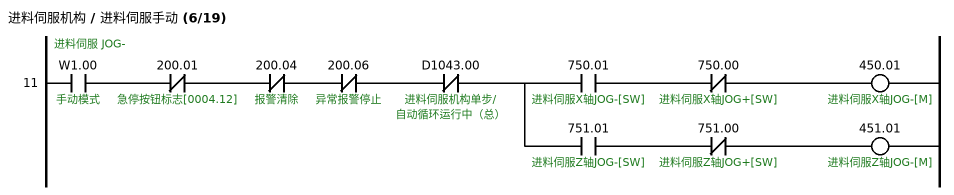
; rung 11: 进料伺服 JOG-
LD W1.00  ; 手动模式
ANDNOT 200.01  ; 急停按钮标志[0004.12]
ANDNOT 200.04  ; 报警清除
ANDNOT 200.06  ; 异常报警停止
ANDNOT D1043.00  ; 进料伺服机构单步/自动循环运行中（总）
OUT TR0
AND 750.01  ; 进料伺服X轴JOG-[SW]
ANDNOT 750.00  ; 进料伺服X轴JOG+[SW]
OUT 450.01  ; 进料伺服X轴JOG-[M]
LD TR0
AND 751.01  ; 进料伺服Z轴JOG-[SW]
ANDNOT 751.00  ; 进料伺服Z轴JOG+[SW]
OUT 451.01  ; 进料伺服Z轴JOG-[M]

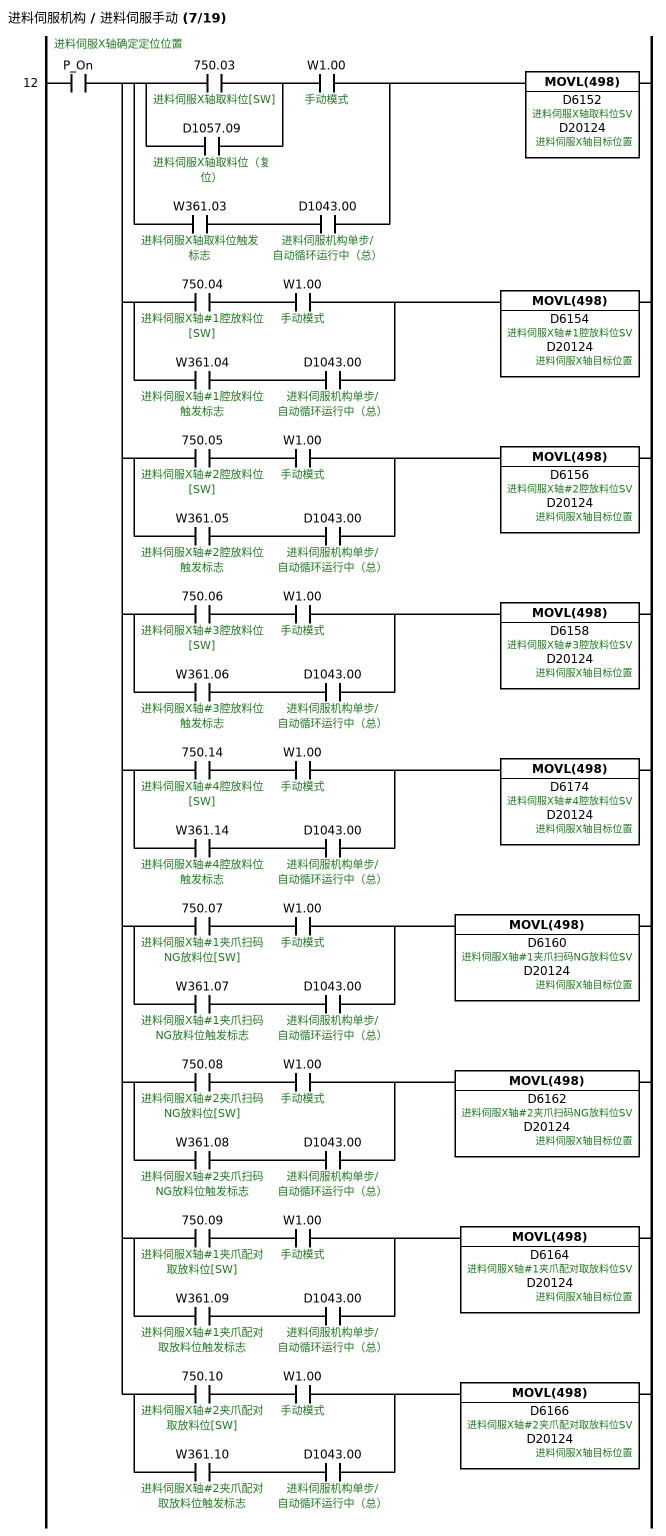
; rung 12: 进料伺服X轴确定定位位置
LD P_On
OUT TR0
LD 750.03  ; 进料伺服X轴取料位[SW]
OR D1057.09  ; 进料伺服X轴取料位（复位）
AND W1.00  ; 手动模式
LD W361.03  ; 进料伺服X轴取料位触发标志
AND D1043.00  ; 进料伺服机构单步/自动循环运行中（总）
ORLD
ANDLD
MOVL(498) D6152 D20124  ; 进料伺服X轴取料位SV, 进料伺服X轴目标位置
LD TR0
LD 750.04  ; 进料伺服X轴#1腔放料位[SW]
AND W1.00  ; 手动模式
LD W361.04  ; 进料伺服X轴#1腔放料位触发标志
AND D1043.00  ; 进料伺服机构单步/自动循环运行中（总）
ORLD
ANDLD
MOVL(498) D6154 D20124  ; 进料伺服X轴#1腔放料位SV, 进料伺服X轴目标位置
LD TR0
LD 750.05  ; 进料伺服X轴#2腔放料位[SW]
AND W1.00  ; 手动模式
LD W361.05  ; 进料伺服X轴#2腔放料位触发标志
AND D1043.00  ; 进料伺服机构单步/自动循环运行中（总）
ORLD
ANDLD
MOVL(498) D6156 D20124  ; 进料伺服X轴#2腔放料位SV, 进料伺服X轴目标位置
LD TR0
LD 750.06  ; 进料伺服X轴#3腔放料位[SW]
AND W1.00  ; 手动模式
LD W361.06  ; 进料伺服X轴#3腔放料位触发标志
AND D1043.00  ; 进料伺服机构单步/自动循环运行中（总）
ORLD
ANDLD
MOVL(498) D6158 D20124  ; 进料伺服X轴#3腔放料位SV, 进料伺服X轴目标位置
LD TR0
LD 750.14  ; 进料伺服X轴#4腔放料位[SW]
AND W1.00  ; 手动模式
LD W361.14  ; 进料伺服X轴#4腔放料位触发标志
AND D1043.00  ; 进料伺服机构单步/自动循环运行中（总）
ORLD
ANDLD
MOVL(498) D6174 D20124  ; 进料伺服X轴#4腔放料位SV, 进料伺服X轴目标位置
LD TR0
LD 750.07  ; 进料伺服X轴#1夹爪扫码NG放料位[SW]
AND W1.00  ; 手动模式
LD W361.07  ; 进料伺服X轴#1夹爪扫码NG放料位触发标志
AND D1043.00  ; 进料伺服机构单步/自动循环运行中（总）
ORLD
ANDLD
MOVL(498) D6160 D20124  ; 进料伺服X轴#1夹爪扫码NG放料位SV, 进料伺服X轴目标位置
LD TR0
LD 750.08  ; 进料伺服X轴#2夹爪扫码NG放料位[SW]
AND W1.00  ; 手动模式
LD W361.08  ; 进料伺服X轴#2夹爪扫码NG放料位触发标志
AND D1043.00  ; 进料伺服机构单步/自动循环运行中（总）
ORLD
ANDLD
MOVL(498) D6162 D20124  ; 进料伺服X轴#2夹爪扫码NG放料位SV, 进料伺服X轴目标位置
LD TR0
LD 750.09  ; 进料伺服X轴#1夹爪配对取放料位[SW]
AND W1.00  ; 手动模式
LD W361.09  ; 进料伺服X轴#1夹爪配对取放料位触发标志
AND D1043.00  ; 进料伺服机构单步/自动循环运行中（总）
ORLD
ANDLD
MOVL(498) D6164 D20124  ; 进料伺服X轴#1夹爪配对取放料位SV, 进料伺服X轴目标位置
LD TR0
LD 750.10  ; 进料伺服X轴#2夹爪配对取放料位[SW]
AND W1.00  ; 手动模式
LD W361.10  ; 进料伺服X轴#2夹爪配对取放料位触发标志
AND D1043.00  ; 进料伺服机构单步/自动循环运行中（总）
ORLD
ANDLD
MOVL(498) D6166 D20124  ; 进料伺服X轴#2夹爪配对取放料位SV, 进料伺服X轴目标位置

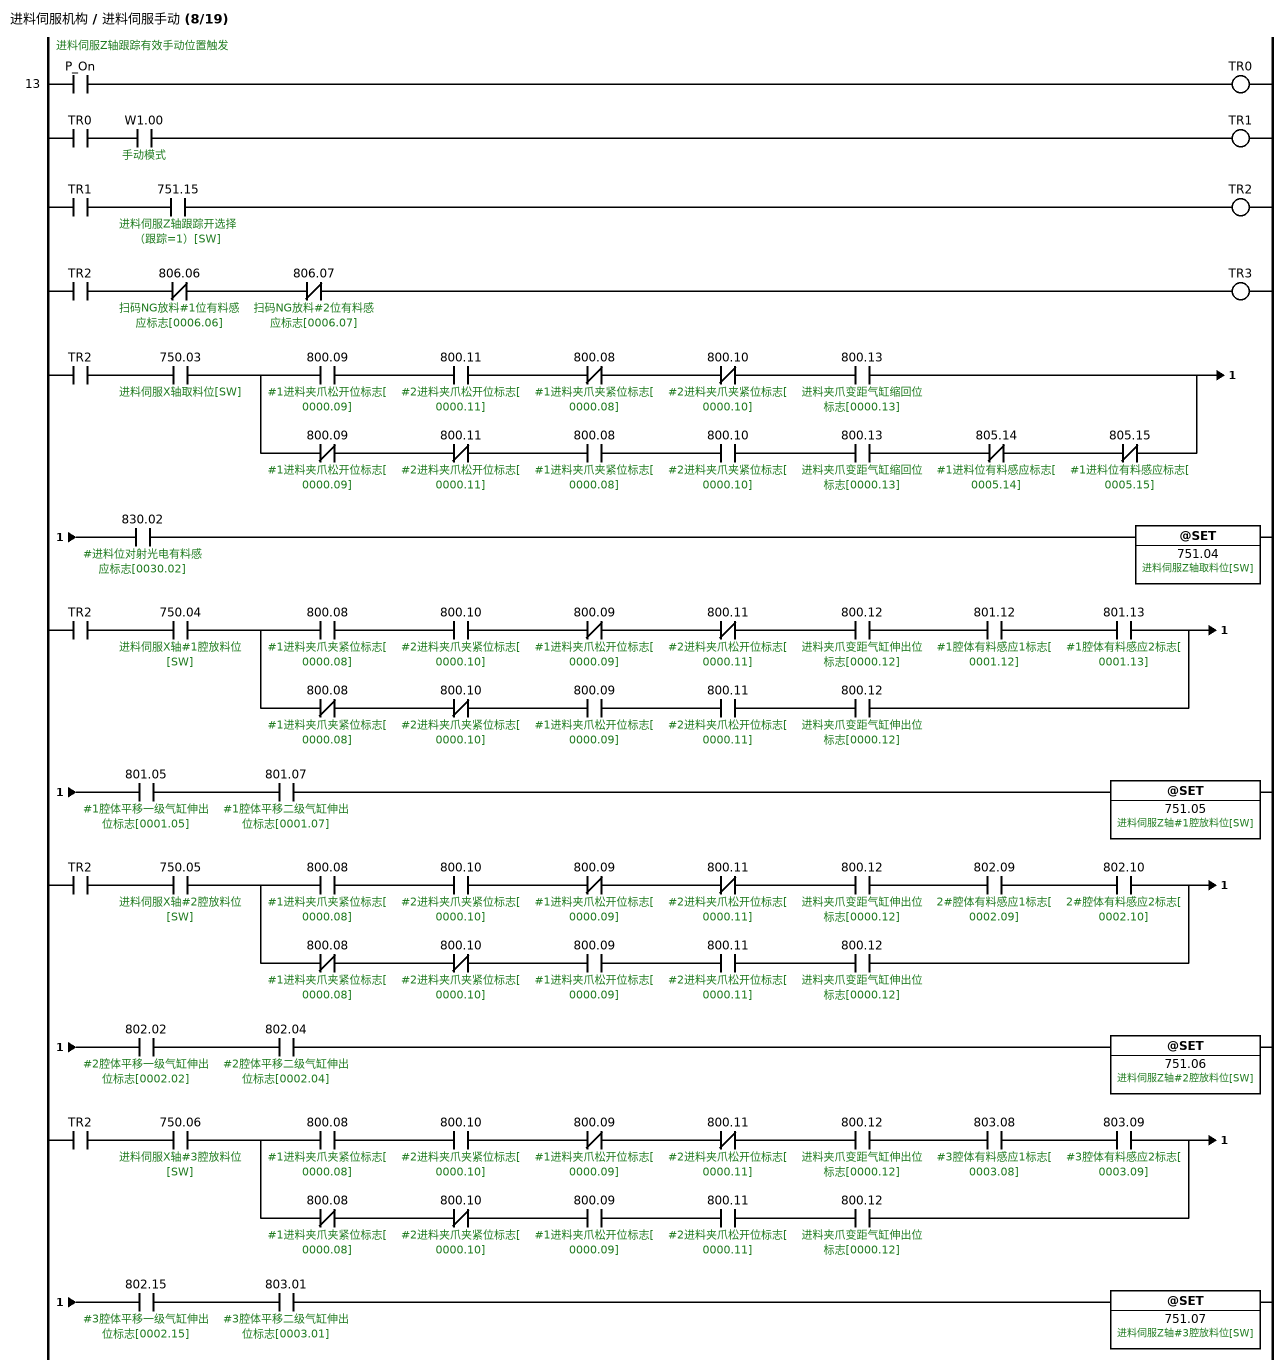

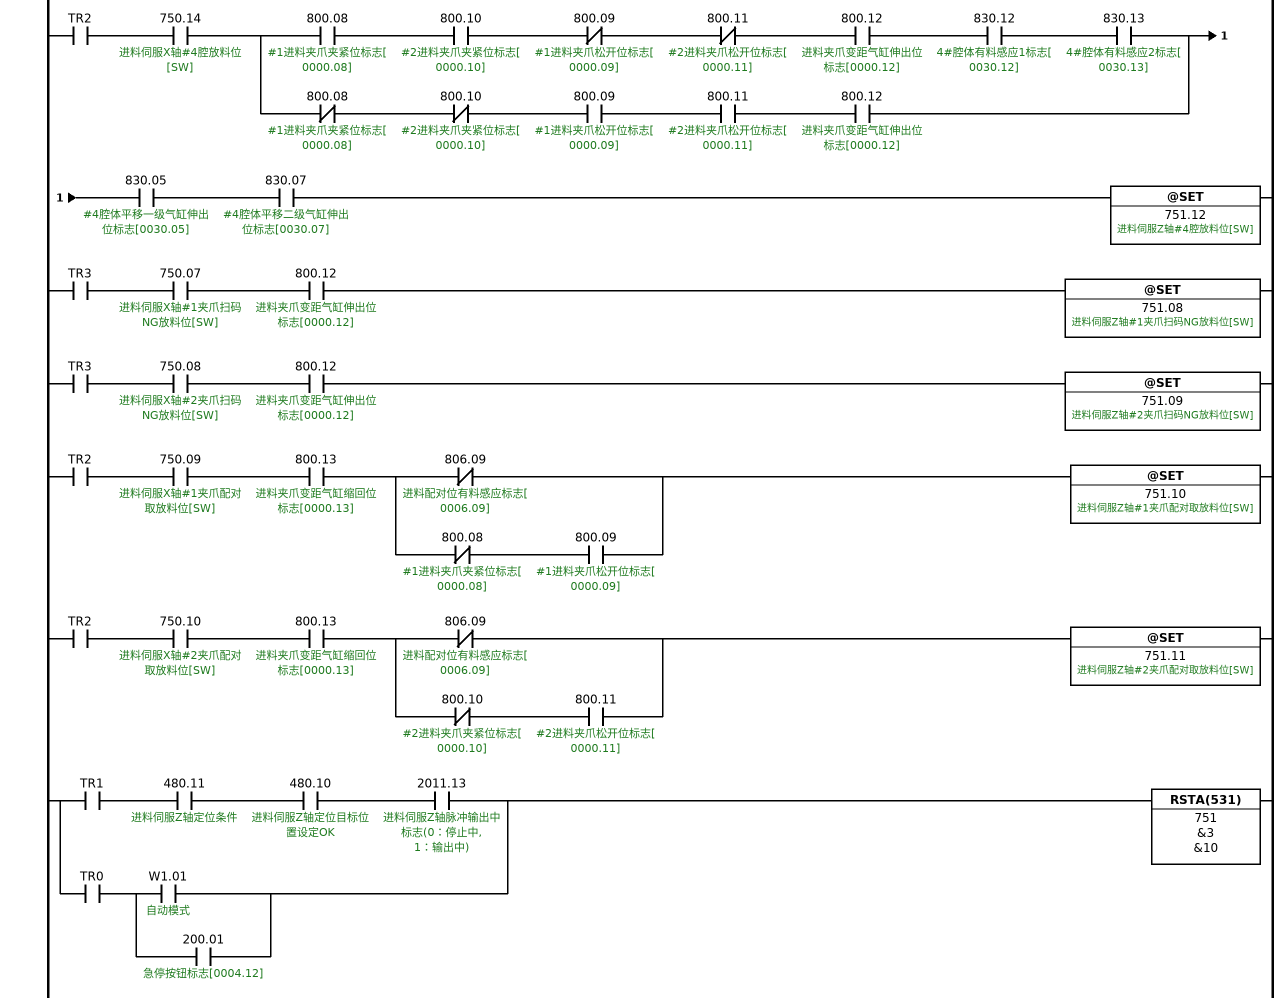
; rung 13: 进料伺服Z轴跟踪有效手动位置触发
LD P_On
OUT TR0
AND W1.00  ; 手动模式
OUT TR1
AND 751.15  ; 进料伺服Z轴跟踪开选择（跟踪=1）[SW]
OUT TR2
AND 750.03  ; 进料伺服X轴取料位[SW]
LD 800.09  ; #1进料夹爪松开位标志[0000.09]
AND 800.11  ; #2进料夹爪松开位标志[0000.11]
ANDNOT 800.08  ; #1进料夹爪夹紧位标志[0000.08]
ANDNOT 800.10  ; #2进料夹爪夹紧位标志[0000.10]
AND 800.13  ; 进料夹爪变距气缸缩回位标志[0000.13]
LDNOT 800.09  ; #1进料夹爪松开位标志[0000.09]
ANDNOT 800.11  ; #2进料夹爪松开位标志[0000.11]
AND 800.08  ; #1进料夹爪夹紧位标志[0000.08]
AND 800.10  ; #2进料夹爪夹紧位标志[0000.10]
AND 800.13  ; 进料夹爪变距气缸缩回位标志[0000.13]
ANDNOT 805.14  ; #1进料位有料感应标志[0005.14]
ANDNOT 805.15  ; #1进料位有料感应标志[0005.15]
ORLD
ANDLD
AND 830.02  ; #进料位对射光电有料感应标志[0030.02]
@SET 751.04  ; 进料伺服Z轴取料位[SW]
LD TR2
AND 750.04  ; 进料伺服X轴#1腔放料位[SW]
LD 800.08  ; #1进料夹爪夹紧位标志[0000.08]
AND 800.10  ; #2进料夹爪夹紧位标志[0000.10]
ANDNOT 800.09  ; #1进料夹爪松开位标志[0000.09]
ANDNOT 800.11  ; #2进料夹爪松开位标志[0000.11]
AND 800.12  ; 进料夹爪变距气缸伸出位标志[0000.12]
AND 801.12  ; #1腔体有料感应1标志[0001.12]
AND 801.13  ; #1腔体有料感应2标志[0001.13]
LDNOT 800.08  ; #1进料夹爪夹紧位标志[0000.08]
ANDNOT 800.10  ; #2进料夹爪夹紧位标志[0000.10]
AND 800.09  ; #1进料夹爪松开位标志[0000.09]
AND 800.11  ; #2进料夹爪松开位标志[0000.11]
AND 800.12  ; 进料夹爪变距气缸伸出位标志[0000.12]
ORLD
ANDLD
AND 801.05  ; #1腔体平移一级气缸伸出位标志[0001.05]
AND 801.07  ; #1腔体平移二级气缸伸出位标志[0001.07]
@SET 751.05  ; 进料伺服Z轴#1腔放料位[SW]
LD TR2
AND 750.05  ; 进料伺服X轴#2腔放料位[SW]
LD 800.08  ; #1进料夹爪夹紧位标志[0000.08]
AND 800.10  ; #2进料夹爪夹紧位标志[0000.10]
ANDNOT 800.09  ; #1进料夹爪松开位标志[0000.09]
ANDNOT 800.11  ; #2进料夹爪松开位标志[0000.11]
AND 800.12  ; 进料夹爪变距气缸伸出位标志[0000.12]
AND 802.09  ; 2#腔体有料感应1标志[0002.09]
AND 802.10  ; 2#腔体有料感应2标志[0002.10]
LDNOT 800.08  ; #1进料夹爪夹紧位标志[0000.08]
ANDNOT 800.10  ; #2进料夹爪夹紧位标志[0000.10]
AND 800.09  ; #1进料夹爪松开位标志[0000.09]
AND 800.11  ; #2进料夹爪松开位标志[0000.11]
AND 800.12  ; 进料夹爪变距气缸伸出位标志[0000.12]
ORLD
ANDLD
AND 802.02  ; #2腔体平移一级气缸伸出位标志[0002.02]
AND 802.04  ; #2腔体平移二级气缸伸出位标志[0002.04]
@SET 751.06  ; 进料伺服Z轴#2腔放料位[SW]
LD TR2
AND 750.06  ; 进料伺服X轴#3腔放料位[SW]
LD 800.08  ; #1进料夹爪夹紧位标志[0000.08]
AND 800.10  ; #2进料夹爪夹紧位标志[0000.10]
ANDNOT 800.09  ; #1进料夹爪松开位标志[0000.09]
ANDNOT 800.11  ; #2进料夹爪松开位标志[0000.11]
AND 800.12  ; 进料夹爪变距气缸伸出位标志[0000.12]
AND 803.08  ; #3腔体有料感应1标志[0003.08]
AND 803.09  ; #3腔体有料感应2标志[0003.09]
LDNOT 800.08  ; #1进料夹爪夹紧位标志[0000.08]
ANDNOT 800.10  ; #2进料夹爪夹紧位标志[0000.10]
AND 800.09  ; #1进料夹爪松开位标志[0000.09]
AND 800.11  ; #2进料夹爪松开位标志[0000.11]
AND 800.12  ; 进料夹爪变距气缸伸出位标志[0000.12]
ORLD
ANDLD
AND 802.15  ; #3腔体平移一级气缸伸出位标志[0002.15]
AND 803.01  ; #3腔体平移二级气缸伸出位标志[0003.01]
@SET 751.07  ; 进料伺服Z轴#3腔放料位[SW]
LD TR2
AND 750.14  ; 进料伺服X轴#4腔放料位[SW]
LD 800.08  ; #1进料夹爪夹紧位标志[0000.08]
AND 800.10  ; #2进料夹爪夹紧位标志[0000.10]
ANDNOT 800.09  ; #1进料夹爪松开位标志[0000.09]
ANDNOT 800.11  ; #2进料夹爪松开位标志[0000.11]
AND 800.12  ; 进料夹爪变距气缸伸出位标志[0000.12]
AND 830.12  ; 4#腔体有料感应1标志[0030.12]
AND 830.13  ; 4#腔体有料感应2标志[0030.13]
LDNOT 800.08  ; #1进料夹爪夹紧位标志[0000.08]
ANDNOT 800.10  ; #2进料夹爪夹紧位标志[0000.10]
AND 800.09  ; #1进料夹爪松开位标志[0000.09]
AND 800.11  ; #2进料夹爪松开位标志[0000.11]
AND 800.12  ; 进料夹爪变距气缸伸出位标志[0000.12]
ORLD
ANDLD
AND 830.05  ; #4腔体平移一级气缸伸出位标志[0030.05]
AND 830.07  ; #4腔体平移二级气缸伸出位标志[0030.07]
@SET 751.12  ; 进料伺服Z轴#4腔放料位[SW]
LD TR2
ANDNOT 806.06  ; 扫码NG放料#1位有料感应标志[0006.06]
ANDNOT 806.07  ; 扫码NG放料#2位有料感应标志[0006.07]
OUT TR3
AND 750.07  ; 进料伺服X轴#1夹爪扫码NG放料位[SW]
AND 800.12  ; 进料夹爪变距气缸伸出位标志[0000.12]
@SET 751.08  ; 进料伺服Z轴#1夹爪扫码NG放料位[SW]
LD TR3
AND 750.08  ; 进料伺服X轴#2夹爪扫码NG放料位[SW]
AND 800.12  ; 进料夹爪变距气缸伸出位标志[0000.12]
@SET 751.09  ; 进料伺服Z轴#2夹爪扫码NG放料位[SW]
LD TR2
AND 750.09  ; 进料伺服X轴#1夹爪配对取放料位[SW]
AND 800.13  ; 进料夹爪变距气缸缩回位标志[0000.13]
LDNOT 806.09  ; 进料配对位有料感应标志[0006.09]
LDNOT 800.08  ; #1进料夹爪夹紧位标志[0000.08]
AND 800.09  ; #1进料夹爪松开位标志[0000.09]
ORLD
ANDLD
@SET 751.10  ; 进料伺服Z轴#1夹爪配对取放料位[SW]
LD TR2
AND 750.10  ; 进料伺服X轴#2夹爪配对取放料位[SW]
AND 800.13  ; 进料夹爪变距气缸缩回位标志[0000.13]
LDNOT 806.09  ; 进料配对位有料感应标志[0006.09]
LDNOT 800.10  ; #2进料夹爪夹紧位标志[0000.10]
AND 800.11  ; #2进料夹爪松开位标志[0000.11]
ORLD
ANDLD
@SET 751.11  ; 进料伺服Z轴#2夹爪配对取放料位[SW]
LD TR1
AND 480.11  ; 进料伺服Z轴定位条件
AND 480.10  ; 进料伺服Z轴定位目标位置设定OK
AND 2011.13  ; 进料伺服Z轴脉冲输出中标志(0：停止中,1：输出中)
LD TR0
LD W1.01  ; 自动模式
OR 200.01  ; 急停按钮标志[0004.12]
ANDLD
ORLD
RSTA(531) 751 &3 &10

